C01819=1084.866,371.145,-96.496,176.864,26.563,154.394
C01820=1084.871,371.355,-96.527,176.867,26.567,154.395
C01821=1084.877,371.565,-96.559,176.870,26.572,154.396
C01822=1084.882,371.775,-96.590,176.873,26.578,154.397
C01823=1084.888,372.022,-96.627,176.876,26.584,154.398
C01824=1084.894,372.269,-96.664,176.880,26.590,154.399
C01825=1084.900,372.516,-96.701,176.883,26.596,154.400
C01826=1084.906,372.763,-96.738,176.886,26.603,154.401
C01827=1084.913,373.011,-96.775,176.890,26.609,154.403
C01828=1084.919,373.257,-96.812,176.892,26.615,154.404
C01829=1084.925,373.504,-96.849,176.896,26.621,154.405
C01830=1084.932,373.752,-96.885,176.900,26.627,154.406
C01831=1084.937,373.998,-96.923,176.902,26.633,154.407
C01832=1084.943,374.246,-96.960,176.906,26.640,154.408
C01833=1084.949,374.493,-96.997,176.909,26.646,154.409
C01834=1084.956,374.740,-97.035,176.913,26.652,154.410
C01835=1084.962,374.988,-97.072,176.916,26.658,154.412
C01836=1084.968,375.234,-97.109,176.919,26.665,154.413
C01837=1084.974,375.481,-97.146,176.923,26.672,154.414
C01838=1084.980,375.728,-97.184,176.925,26.678,154.415
C01839=1084.986,375.975,-97.220,176.929,26.684,154.416
C01840=1084.993,376.223,-97.258,176.933,26.690,154.417
C01841=1084.998,376.469,-97.296,176.936,26.697,154.418
C01842=1085.004,376.717,-97.333,176.939,26.703,154.420
C01843=1085.011,376.963,-97.370,176.942,26.709,154.421
C01844=1085.016,377.210,-97.407,176.946,26.716,154.422
C01845=1085.023,377.458,-97.445,176.948,26.722,154.423
C01846=1085.029,377.705,-97.483,176.952,26.729,154.424
C01847=1085.035,377.952,-97.520,176.955,26.736,154.426
C01848=1085.041,378.198,-97.557,176.959,26.742,154.427
C01849=1085.047,378.446,-97.595,176.962,26.748,154.428
C01850=1085.053,378.693,-97.633,176.965,26.755,154.429
C01851=1085.060,378.940,-97.670,176.969,26.761,154.430
C01852=1085.066,379.187,-97.708,176.972,26.768,154.431
C01853=1085.072,379.434,-97.745,176.976,26.775,154.433
C01854=1085.078,379.681,-97.783,176.979,26.781,154.434
C01855=1085.084,379.928,-97.821,176.982,26.788,154.435
C01856=1085.091,380.174,-97.859,176.986,26.795,154.436
C01857=1085.097,380.422,-97.896,176.989,26.801,154.438
C01858=1085.103,380.669,-97.934,176.993,26.808,154.439
C01859=1085.109,380.916,-97.971,176.995,26.814,154.440
C01860=1085.115,381.163,-98.009,176.999,26.821,154.441
C01861=1085.122,381.410,-98.047,177.002,26.828,154.443
C01862=1085.128,381.657,-98.084,177.006,26.834,154.444
C01863=1085.135,381.904,-98.123,177.009,26.841,154.445
C01864=1085.141,382.151,-98.160,177.012,26.847,154.446
C01865=1085.147,382.398,-98.198,177.016,26.854,154.447
C01866=1085.153,382.645,-98.236,177.019,26.861,154.449
C01867=1085.159,382.891,-98.275,177.022,26.868,154.450
C01868=1085.165,383.138,-98.312,177.026,26.875,154.451
C01869=1085.172,383.385,-98.351,177.030,26.882,154.453
C01870=1085.178,383.632,-98.388,177.032,26.888,154.454
C01871=1085.182,383.856,-98.423,177.036,26.895,154.455
C01872=1085.188,384.080,-98.458,177.038,26.901,154.456
C01873=1085.194,384.304,-98.492,177.042,26.908,154.457
C01874=1085.199,384.527,-98.527,177.045,26.914,154.459
C01875=1085.205,384.752,-98.562,177.047,26.920,154.460
C01876=1085.211,384.975,-98.596,177.051,26.926,154.461
C01877=1085.217,385.199,-98.631,177.054,26.932,154.462
C01878=1085.222,385.423,-98.666,177.057,26.939,154.463
C01879=1085.228,385.671,-98.704,177.061,26.946,154.465
C01880=1085.234,385.917,-98.742,177.063,26.953,154.466
C01881=1085.241,386.164,-98.780,177.067,26.960,154.467
C01882=1085.247,386.410,-98.819,177.070,26.967,154.469
C01883=1085.254,386.658,-98.857,177.074,26.974,154.470
C01884=1085.260,386.904,-98.895,177.077,26.981,154.471
C01885=1085.266,387.152,-98.934,177.081,26.988,154.473
C01886=1085.271,387.399,-98.972,177.084,26.995,154.474
C01887=1085.278,387.645,-99.011,177.088,27.003,154.475
C01888=1085.284,387.891,-99.049,177.091,27.010,154.477
C01889=1085.291,388.139,-99.087,177.095,27.017,154.478
C01890=1085.296,388.385,-99.126,177.098,27.024,154.479
C01891=1085.303,388.633,-99.165,177.101,27.031,154.481
C01892=1085.310,388.880,-99.203,177.105,27.038,154.482
C01893=1085.316,389.126,-99.242,177.108,27.045,154.484
C01894=1085.322,389.373,-99.280,177.111,27.053,154.485
C01895=1085.328,389.620,-99.319,177.114,27.060,154.486
C01896=1085.335,389.866,-99.358,177.118,27.067,154.488
C01897=1085.341,390.114,-99.396,177.121,27.075,154.489
C01898=1085.347,390.360,-99.434,177.125,27.082,154.491
C01899=1085.354,390.607,-99.474,177.128,27.089,154.492
C01900=1085.360,390.854,-99.513,177.132,27.096,154.493
C01901=1085.367,391.100,-99.551,177.135,27.104,154.495
C01902=1085.372,391.348,-99.590,177.139,27.111,154.496
C01903=1085.379,391.595,-99.629,177.142,27.119,154.498
C01904=1085.386,391.841,-99.668,177.146,27.126,154.499
C01905=1085.391,392.088,-99.707,177.149,27.133,154.500
C01906=1085.398,392.335,-99.746,177.152,27.141,154.502
C01907=1085.404,392.582,-99.785,177.156,27.148,154.503
C01908=1085.411,392.828,-99.823,177.159,27.156,154.505
C01909=1085.417,393.075,-99.863,177.163,27.163,154.506
C01910=1085.423,393.322,-99.902,177.166,27.171,154.508
C01911=1085.429,393.569,-99.941,177.170,27.179,154.509
C01912=1085.436,393.815,-99.980,177.173,27.186,154.511
C01913=1085.442,394.062,-100.019,177.176,27.194,154.512
C01914=1085.449,394.309,-100.058,177.180,27.201,154.514
C01915=1085.455,394.556,-100.097,177.183,27.209,154.515
C01916=1085.461,394.803,-100.136,177.187,27.217,154.517
C01917=1085.467,395.049,-100.176,177.191,27.225,154.518
C01918=1085.474,395.296,-100.215,177.194,27.232,154.520
C01919=1085.480,395.543,-100.254,177.198,27.240,154.521
C01920=1085.486,395.790,-100.294,177.201,27.248,154.523
C01921=1085.493,396.037,-100.332,177.205,27.256,154.524
C01922=1085.499,396.283,-100.373,177.208,27.264,154.526
C01923=1085.505,396.530,-100.412,177.211,27.271,154.527
C01924=1085.511,396.777,-100.451,177.215,27.279,154.529
C01925=1085.518,397.023,-100.491,177.218,27.287,154.530
C01926=1085.524,397.270,-100.530,177.222,27.295,154.532
C01927=1085.530,397.501,-100.566,177.225,27.302,154.533
C01928=1085.536,397.732,-100.604,177.229,27.310,154.535
C01929=1085.542,397.963,-100.640,177.231,27.317,154.536
C01930=1085.548,398.194,-100.678,177.235,27.325,154.538
C01931=1085.554,398.424,-100.715,177.238,27.332,154.539
C01932=1085.560,398.655,-100.752,177.242,27.339,154.541
C01933=1085.566,398.886,-100.789,177.245,27.347,154.542
C01934=1085.572,399.116,-100.826,177.248,27.354,154.544
C01935=1085.578,399.363,-100.866,177.252,27.363,154.545
C01936=1085.585,399.610,-100.905,177.255,27.371,154.547
C01937=1085.591,399.856,-100.945,177.258,27.379,154.549
C01938=1085.597,400.103,-100.985,177.262,27.387,154.550
C01939=1085.604,400.350,-101.025,177.265,27.395,154.552
C01940=1085.610,400.596,-101.065,177.269,27.404,154.553
C01941=1085.616,400.844,-101.104,177.272,27.411,154.555
C01942=1085.622,401.090,-101.145,177.276,27.420,154.557
C01943=1085.629,401.337,-101.185,177.280,27.428,154.558
C01944=1085.635,401.584,-101.224,177.283,27.437,154.560
C01945=1085.641,401.830,-101.264,177.286,27.445,154.562
C01946=1085.648,402.077,-101.305,177.290,27.453,154.563
C01947=1085.655,402.324,-101.345,177.294,27.462,154.565
C01948=1085.661,402.571,-101.385,177.297,27.470,154.567
C01949=1085.667,402.817,-101.425,177.301,27.478,154.568
C01950=1085.673,403.064,-101.465,177.304,27.487,154.570
C01951=1085.680,403.311,-101.505,177.308,27.495,154.572
C01952=1085.686,403.557,-101.545,177.312,27.504,154.573
C01953=1085.693,403.804,-101.585,177.315,27.512,154.575
C01954=1085.700,404.051,-101.626,177.318,27.521,154.577
C01955=1085.706,404.297,-101.666,177.323,27.529,154.579
C01956=1085.712,404.544,-101.706,177.326,27.537,154.580
C01957=1085.719,404.790,-101.746,177.329,27.546,154.582
C01958=1085.725,405.037,-101.786,177.333,27.555,154.584
C01959=1085.731,405.283,-101.826,177.337,27.564,154.586
C01960=1085.738,405.531,-101.867,177.340,27.572,154.587
C01961=1085.745,405.777,-101.908,177.343,27.581,154.589
C01962=1085.751,406.023,-101.949,177.348,27.590,154.591
C01963=1085.757,406.270,-101.989,177.351,27.598,154.593
C01964=1085.764,406.517,-102.029,177.354,27.607,154.594
C01965=1085.771,406.764,-102.069,177.359,27.616,154.596
C01966=1085.776,407.010,-102.111,177.362,27.625,154.598
C01967=1085.783,407.256,-102.151,177.365,27.634,154.600
C01968=1085.790,407.504,-102.191,177.369,27.643,154.602
C01969=1085.797,407.750,-102.232,177.373,27.652,154.604
C01970=1085.802,407.996,-102.273,177.376,27.660,154.605
C01971=1085.809,408.244,-102.314,177.380,27.669,154.607
C01972=1085.815,408.490,-102.355,177.383,27.679,154.609
C01973=1085.821,408.736,-102.395,177.388,27.688,154.611
C01974=1085.828,408.982,-102.436,177.391,27.697,154.613
C01975=1085.834,409.230,-102.477,177.394,27.705,154.615
C01976=1085.841,409.476,-102.518,177.399,27.715,154.616
C01977=1085.847,409.722,-102.559,177.402,27.724,154.618
C01978=1085.854,409.969,-102.600,177.406,27.733,154.620
C01979=1085.860,410.216,-102.640,177.409,27.742,154.622
C01980=1085.867,410.462,-102.682,177.413,27.751,154.624
C01981=1085.874,410.708,-102.723,177.417,27.761,154.626
C01982=1085.879,410.955,-102.764,177.420,27.770,154.628
C01983=1085.886,411.187,-102.802,177.424,27.779,154.630
C01984=1085.892,411.418,-102.841,177.428,27.788,154.631
C01985=1085.898,411.649,-102.879,177.431,27.796,154.633
C01986=1085.904,411.882,-102.918,177.434,27.805,154.635
C01987=1085.910,412.113,-102.956,177.438,27.814,154.637
C01988=1085.917,412.344,-102.996,177.441,27.822,154.639
C01989=1085.923,412.576,-103.035,177.444,27.832,154.641
C01990=1085.929,412.807,-103.072,177.449,27.841,154.642
C01991=1085.935,413.054,-103.114,177.452,27.850,154.644
C01992=1085.942,413.300,-103.155,177.456,27.859,154.646
C01993=1085.948,413.547,-103.197,177.459,27.869,154.648
C01994=1085.956,413.793,-103.238,177.464,27.878,154.650
C01995=1085.962,414.040,-103.280,177.467,27.888,154.652
C01996=1085.969,414.286,-103.321,177.471,27.897,154.654
C01997=1085.975,414.532,-103.362,177.475,27.907,154.656
C01998=1085.982,414.779,-103.404,177.479,27.917,154.658
C01999=1085.988,415.025,-103.445,177.483,27.926,154.660
C02000=1085.995,415.272,-103.487,177.486,27.936,154.662
C02001=1086.002,415.519,-103.528,177.490,27.946,154.664
C02002=1086.008,415.765,-103.570,177.494,27.956,154.666
C02003=1086.015,416.011,-103.611,177.498,27.966,154.668
C02004=1086.022,416.258,-103.653,177.502,27.976,154.671
C02005=1086.028,416.504,-103.695,177.505,27.985,154.673
C02006=1086.035,416.751,-103.737,177.509,27.996,154.675
C02007=1086.041,416.997,-103.779,177.513,28.005,154.677
C02008=1086.048,417.243,-103.820,177.517,28.016,154.679
C02009=1086.055,417.490,-103.862,177.521,28.025,154.681
C02010=1086.061,417.736,-103.904,177.525,28.036,154.683
C02011=1086.067,417.983,-103.946,177.529,28.046,154.685
C02012=1086.074,418.229,-103.988,177.532,28.056,154.687
C02013=1086.080,418.475,-104.030,177.536,28.066,154.690
C02014=1086.087,418.721,-104.072,177.541,28.076,154.692
C02015=1086.094,418.968,-104.114,177.544,28.086,154.694
C02016=1086.101,419.214,-104.156,177.548,28.097,154.696
C02017=1086.107,419.460,-104.198,177.552,28.107,154.698
C02018=1086.114,419.707,-104.240,177.556,28.117,154.700
C02019=1086.121,419.954,-104.282,177.560,28.127,154.703
C02020=1086.127,420.200,-104.324,177.564,28.138,154.705
C02021=1086.134,420.445,-104.367,177.568,28.149,154.707
C02022=1086.140,420.692,-104.408,177.572,28.159,154.709
C02023=1086.147,420.939,-104.451,177.575,28.169,154.711
C02024=1086.154,421.185,-104.494,177.579,28.180,154.714
C02025=1086.162,421.431,-104.535,177.583,28.190,154.716
C02026=1086.168,421.677,-104.578,177.588,28.201,154.718
C02027=1086.174,421.923,-104.619,177.592,28.211,154.720
C02028=1086.181,422.170,-104.662,177.596,28.222,154.723
C02029=1086.188,422.416,-104.705,177.599,28.233,154.725
C02030=1086.194,422.663,-104.748,177.603,28.244,154.727
C02031=1086.201,422.909,-104.790,177.607,28.254,154.730
C02032=1086.208,423.155,-104.833,177.611,28.265,154.732
C02033=1086.215,423.401,-104.875,177.616,28.276,154.734
C02034=1086.221,423.647,-104.917,177.620,28.287,154.737
C02035=1086.228,423.893,-104.960,177.624,28.298,154.739
C02036=1086.234,424.140,-105.003,177.627,28.309,154.741
C02037=1086.241,424.386,-105.046,177.631,28.319,154.744
C02038=1086.248,424.632,-105.089,177.635,28.331,154.746
C02039=1086.259,425.045,-105.160,177.642,28.349,154.750
C02040=1086.271,425.458,-105.232,177.649,28.368,154.754
C02041=1086.282,425.871,-105.304,177.656,28.386,154.758
C02042=1086.293,426.284,-105.376,177.663,28.405,154.762
C02043=1086.300,426.529,-105.419,177.667,28.417,154.765
C02044=1086.307,426.775,-105.462,177.671,28.428,154.767
C02045=1086.313,427.022,-105.505,177.675,28.439,154.769
C02046=1086.320,427.268,-105.548,177.679,28.450,154.772
C02047=1086.327,427.514,-105.591,177.683,28.462,154.774
C02048=1086.334,427.760,-105.634,177.687,28.473,154.777
C02049=1086.341,428.006,-105.678,177.691,28.485,154.779
C02050=1086.348,428.253,-105.721,177.695,28.496,154.782
C02051=1086.356,428.498,-105.764,177.700,28.507,154.784
C02052=1086.362,428.745,-105.807,177.704,28.519,154.787
C02053=1086.369,428.991,-105.851,177.709,28.531,154.789
C02054=1086.375,429.237,-105.894,177.713,28.543,154.792
C02055=1086.382,429.482,-105.938,177.717,28.555,154.795
C02056=1086.389,429.729,-105.981,177.721,28.566,154.797
C02057=1086.396,429.974,-106.024,177.725,28.578,154.800
C02058=1086.403,430.221,-106.068,177.729,28.590,154.802
C02059=1086.410,430.467,-106.112,177.733,28.602,154.805
C02060=1086.416,430.713,-106.155,177.737,28.614,154.808
C02061=1086.423,430.958,-106.199,177.741,28.626,154.810
C02062=1086.430,431.204,-106.243,177.746,28.638,154.813
C02063=1086.437,431.451,-106.287,177.751,28.650,154.815
C02064=1086.444,431.697,-106.330,177.755,28.662,154.818
C02065=1086.450,431.943,-106.374,177.759,28.674,154.821
C02066=1086.458,432.188,-106.417,177.763,28.686,154.823
C02067=1086.465,432.435,-106.461,177.767,28.698,154.826
C02068=1086.472,432.681,-106.505,177.772,28.710,154.829
C02069=1086.478,432.927,-106.548,177.776,28.723,154.832
C02070=1086.485,433.173,-106.593,177.780,28.735,154.834
C02071=1086.492,433.419,-106.637,177.784,28.748,154.837
C02072=1086.499,433.664,-106.680,177.789,28.760,154.840
C02073=1086.506,433.911,-106.725,177.793,28.773,154.843
C02074=1086.513,434.156,-106.769,177.797,28.785,154.845
C02075=1086.521,434.468,-106.825,177.803,28.801,154.849
C02076=1086.530,434.780,-106.881,177.808,28.817,154.852
C02077=1086.539,435.092,-106.937,177.814,28.833,154.856
C02078=1086.548,435.404,-106.993,177.820,28.849,154.860
C02079=1086.555,435.649,-107.037,177.824,28.862,154.862
C02080=1086.561,435.895,-107.081,177.829,28.875,154.865
C02081=1086.569,436.141,-107.126,177.833,28.888,154.868
C02082=1086.575,436.387,-107.171,177.837,28.901,154.871
C02083=1086.583,436.633,-107.214,177.842,28.914,154.874
C02084=1086.590,436.878,-107.259,177.846,28.926,154.877
C02085=1086.597,437.124,-107.304,177.850,28.939,154.880
C02086=1086.604,437.370,-107.349,177.855,28.953,154.883
C02087=1086.611,437.616,-107.393,177.859,28.966,154.886
C02088=1086.618,437.862,-107.437,177.864,28.979,154.888
C02089=1086.625,438.108,-107.482,177.868,28.992,154.891
C02090=1086.632,438.353,-107.527,177.872,29.005,154.894
C02091=1086.639,438.584,-107.568,177.876,29.018,154.897
C02092=1086.646,438.814,-107.610,177.881,29.030,154.900
C02093=1086.652,439.044,-107.653,177.886,29.043,154.903
C02094=1086.658,439.274,-107.694,177.890,29.056,154.906
C02095=1086.666,439.505,-107.737,177.894,29.068,154.909
C02096=1086.672,439.735,-107.778,177.898,29.081,154.911
C02097=1086.679,439.966,-107.821,177.902,29.093,154.914
C02098=1086.686,440.196,-107.863,177.907,29.106,154.917
C02099=1086.693,440.442,-107.908,177.911,29.120,154.920
C02100=1086.700,440.687,-107.953,177.916,29.134,154.923
C02101=1086.707,440.933,-107.998,177.920,29.147,154.926
C02102=1086.715,441.179,-108.043,177.925,29.161,154.930
C02103=1086.721,441.424,-108.088,177.930,29.175,154.933
C02104=1086.728,441.670,-108.133,177.934,29.189,154.936
C02105=1086.736,441.916,-108.179,177.939,29.203,154.939
C02106=1086.743,442.162,-108.224,177.943,29.217,154.942
C02107=1086.750,442.407,-108.268,177.948,29.231,154.945
C02108=1086.756,442.653,-108.315,177.952,29.245,154.949
C02109=1086.764,442.898,-108.360,177.957,29.260,154.952
C02110=1086.771,443.144,-108.405,177.962,29.274,154.955
C02111=1086.778,443.389,-108.451,177.966,29.288,154.958
C02112=1086.785,443.635,-108.496,177.971,29.302,154.962
C02113=1086.793,443.881,-108.542,177.976,29.317,154.965
C02114=1086.800,444.127,-108.588,177.980,29.331,154.968
C02115=1086.807,444.373,-108.633,177.985,29.346,154.972
C02116=1086.815,444.618,-108.679,177.991,29.360,154.975
C02117=1086.821,444.863,-108.724,177.995,29.374,154.978
C02118=1086.829,445.109,-108.770,178.000,29.389,154.981
C02119=1086.836,445.354,-108.816,178.004,29.404,154.985
C02120=1086.843,445.600,-108.862,178.008,29.418,154.988
C02121=1086.851,445.845,-108.908,178.012,29.433,154.992
C02122=1086.858,446.091,-108.954,178.016,29.448,154.995
C02123=1086.865,446.336,-108.999,178.019,29.462,154.999
C02124=1086.872,446.582,-109.046,178.022,29.477,155.002
C02125=1086.880,446.828,-109.091,178.025,29.491,155.005
C02126=1086.887,447.073,-109.138,178.029,29.506,155.009
C02127=1086.894,447.319,-109.183,178.032,29.520,155.012
C02128=1086.901,447.565,-109.229,178.034,29.535,155.016
C02129=1086.908,447.810,-109.276,178.036,29.549,155.019
C02130=1086.916,448.056,-109.321,178.038,29.563,155.023
C02131=1086.923,448.301,-109.368,178.040,29.578,155.027
C02132=1086.931,448.546,-109.414,178.043,29.593,155.030
C02133=1086.938,448.793,-109.461,178.044,29.607,155.034
C02134=1086.946,449.038,-109.506,178.045,29.621,155.037
C02135=1086.952,449.283,-109.553,178.046,29.636,155.041
C02136=1086.960,449.527,-109.599,178.048,29.650,155.044
C02137=1086.969,449.773,-109.645,178.049,29.664,155.048
C02138=1086.980,450.019,-109.689,178.050,29.676,155.051
C02139=1086.604,450.011,-109.889,178.013,29.864,155.102
C02140=1086.592,449.765,-109.845,178.012,29.851,155.098
C02141=1086.583,449.520,-109.798,178.010,29.837,155.095
C02142=1086.576,449.275,-109.753,178.009,29.823,155.091
C02143=1086.568,449.031,-109.707,178.007,29.808,155.088
C02144=1086.561,448.785,-109.661,178.006,29.794,155.084
C02145=1086.554,448.540,-109.614,178.005,29.780,155.081
C02146=1086.546,448.294,-109.568,178.002,29.765,155.077
C02147=1086.539,448.048,-109.521,178.000,29.750,155.074
C02148=1086.531,447.803,-109.475,177.998,29.736,155.070
C02149=1086.524,447.557,-109.429,177.995,29.721,155.066
C02150=1086.516,447.312,-109.383,177.993,29.707,155.063
C02151=1086.510,447.066,-109.337,177.990,29.693,155.060
C02152=1086.503,446.820,-109.291,177.987,29.678,155.056
C02153=1086.495,446.576,-109.244,177.983,29.663,155.053
C02154=1086.488,446.330,-109.198,177.980,29.649,155.049
C02155=1086.480,446.084,-109.152,177.977,29.634,155.046
C02156=1086.473,445.839,-109.106,177.973,29.619,155.042
C02157=1086.466,445.593,-109.060,177.969,29.605,155.039
C02158=1086.459,445.347,-109.014,177.964,29.590,155.035
C02159=1086.451,445.102,-108.969,177.960,29.576,155.032
C02160=1086.443,444.857,-108.923,177.955,29.561,155.029
C02161=1086.437,444.611,-108.877,177.950,29.546,155.025
C02162=1086.429,444.365,-108.832,177.946,29.532,155.022
C02163=1086.422,444.119,-108.786,177.941,29.517,155.019
C02164=1086.415,443.874,-108.740,177.935,29.503,155.015
C02165=1086.407,443.628,-108.694,177.931,29.489,155.012
C02166=1086.401,443.383,-108.648,177.926,29.474,155.009
C02167=1086.393,443.137,-108.603,177.921,29.460,155.005
C02168=1086.386,442.892,-108.558,177.917,29.446,155.002
C02169=1086.378,442.646,-108.513,177.912,29.431,154.999
C02170=1086.372,442.400,-108.467,177.907,29.417,154.996
C02171=1086.365,442.155,-108.421,177.902,29.403,154.993
C02172=1086.357,441.909,-108.376,177.897,29.389,154.989
C02173=1086.350,441.664,-108.331,177.893,29.375,154.986
C02174=1086.343,441.417,-108.285,177.888,29.361,154.983
C02175=1086.336,441.172,-108.241,177.884,29.347,154.980
C02176=1086.329,440.927,-108.195,177.879,29.333,154.977
C02177=1086.321,440.680,-108.150,177.874,29.320,154.974
C02178=1086.314,440.434,-108.105,177.869,29.306,154.971
C02179=1086.307,440.190,-108.060,177.865,29.292,154.967
C02180=1086.301,439.966,-108.018,177.861,29.280,154.965
C02181=1086.294,439.742,-107.978,177.857,29.267,154.962
C02182=1086.288,439.519,-107.937,177.852,29.255,154.959
C02183=1086.281,439.295,-107.896,177.848,29.243,154.956
C02184=1086.275,439.072,-107.855,177.844,29.231,154.954
C02185=1086.267,438.849,-107.815,177.839,29.218,154.951
C02186=1086.261,438.626,-107.774,177.836,29.206,154.948
C02187=1086.255,438.402,-107.733,177.832,29.194,154.945
C02188=1086.247,438.156,-107.688,177.826,29.181,154.942
C02189=1086.241,437.911,-107.644,177.822,29.168,154.939
C02190=1086.233,437.665,-107.599,177.818,29.155,154.936
C02191=1086.227,437.420,-107.554,177.813,29.141,154.933
C02192=1086.220,437.173,-107.510,177.809,29.128,154.931
C02193=1086.212,436.927,-107.465,177.804,29.115,154.928
C02194=1086.206,436.681,-107.421,177.800,29.102,154.925
C02195=1086.199,436.436,-107.376,177.795,29.089,154.922
C02196=1086.191,436.190,-107.333,177.790,29.076,154.919
C02197=1086.184,435.944,-107.288,177.786,29.063,154.916
C02198=1086.177,435.698,-107.243,177.782,29.050,154.913
C02199=1086.171,435.452,-107.199,177.777,29.037,154.910
C02200=1086.163,435.206,-107.154,177.773,29.025,154.907
C02201=1086.157,434.961,-107.110,177.768,29.012,154.905
C02202=1086.150,434.714,-107.065,177.764,28.999,154.902
C02203=1086.142,434.469,-107.021,177.759,28.987,154.899
C02204=1086.136,434.223,-106.978,177.755,28.974,154.896
C02205=1086.129,433.977,-106.933,177.751,28.961,154.893
C02206=1086.122,433.731,-106.889,177.747,28.949,154.891
C02207=1086.115,433.485,-106.845,177.742,28.936,154.888
C02208=1086.107,433.240,-106.801,177.738,28.924,154.885
C02209=1086.101,432.994,-106.757,177.733,28.912,154.882
C02210=1086.095,432.748,-106.713,177.729,28.899,154.880
C02211=1086.088,432.501,-106.669,177.725,28.887,154.877
C02212=1086.080,432.255,-106.626,177.720,28.875,154.874
C02213=1086.074,432.010,-106.581,177.716,28.863,154.872
C02214=1086.066,431.764,-106.537,177.712,28.851,154.869
C02215=1086.059,431.518,-106.493,177.707,28.838,154.866
C02216=1086.052,431.272,-106.450,177.703,28.826,154.863
C02217=1086.045,431.025,-106.406,177.699,28.815,154.861
C02218=1086.039,430.779,-106.362,177.694,28.802,154.858
C02219=1086.032,430.534,-106.319,177.690,28.790,154.856
C02220=1086.025,430.288,-106.275,177.686,28.778,154.853
C02221=1086.018,430.042,-106.232,177.681,28.766,154.850
C02222=1086.011,429.795,-106.188,177.677,28.755,154.848
C02223=1086.004,429.550,-106.144,177.673,28.743,154.845
C02224=1085.998,429.303,-106.101,177.669,28.731,154.843
C02225=1085.991,429.057,-106.058,177.665,28.720,154.840
C02226=1085.984,428.811,-106.014,177.661,28.708,154.838
C02227=1085.977,428.566,-105.971,177.656,28.696,154.835
C02228=1085.970,428.318,-105.927,177.652,28.685,154.832
C02229=1085.963,428.073,-105.884,177.648,28.673,154.830
C02230=1085.956,427.827,-105.841,177.643,28.661,154.827
C02231=1085.949,427.581,-105.798,177.639,28.650,154.825
C02232=1085.943,427.335,-105.754,177.634,28.639,154.822
C02233=1085.936,427.089,-105.712,177.630,28.627,154.820
C02234=1085.929,426.843,-105.669,177.626,28.616,154.817
C02235=1085.922,426.596,-105.625,177.622,28.604,154.815
C02236=1085.915,426.356,-105.583,177.619,28.593,154.813
C02237=1085.908,426.116,-105.542,177.614,28.582,154.810
C02238=1085.902,425.877,-105.499,177.610,28.571,154.808
C02239=1085.896,425.636,-105.458,177.606,28.561,154.806
C02240=1085.889,425.397,-105.415,177.602,28.549,154.803
C02241=1085.882,425.157,-105.374,177.598,28.539,154.801
C02242=1085.876,424.917,-105.333,177.594,28.528,154.799
C02243=1085.869,424.677,-105.290,177.590,28.517,154.796
C02244=1085.862,424.431,-105.248,177.586,28.506,154.794
C02245=1085.855,424.184,-105.205,177.582,28.495,154.791
C02246=1085.849,423.938,-105.163,177.577,28.484,154.789
C02247=1085.842,423.692,-105.119,177.574,28.473,154.787
C02248=1085.835,423.446,-105.076,177.570,28.462,154.784
C02249=1085.828,423.200,-105.034,177.566,28.452,154.782
C02250=1085.822,422.953,-104.991,177.562,28.441,154.780
C02251=1085.815,422.707,-104.949,177.557,28.430,154.777
C02252=1085.808,422.461,-104.906,177.553,28.419,154.775
C02253=1085.802,422.215,-104.863,177.549,28.408,154.773
C02254=1085.796,421.969,-104.821,177.546,28.398,154.771
C02255=1085.789,421.722,-104.778,177.542,28.387,154.768
C02256=1085.781,421.476,-104.737,177.537,28.376,154.766
C02257=1085.775,421.229,-104.694,177.533,28.366,154.764
C02258=1085.768,420.983,-104.652,177.529,28.355,154.761
C02259=1085.761,420.737,-104.609,177.526,28.345,154.759
C02260=1085.754,420.491,-104.567,177.522,28.334,154.757
C02261=1085.748,420.244,-104.525,177.517,28.324,154.755
C02262=1085.741,419.998,-104.483,177.513,28.314,154.753
C02263=1085.734,419.752,-104.440,177.510,28.303,154.750
C02264=1085.724,419.343,-104.370,177.503,28.286,154.747
C02265=1085.712,418.933,-104.301,177.497,28.269,154.743
C02266=1085.702,418.525,-104.231,177.490,28.252,154.740
C02267=1085.690,418.115,-104.161,177.484,28.235,154.736
C02268=1085.684,417.869,-104.119,177.479,28.225,154.734
C02269=1085.677,417.623,-104.077,177.475,28.215,154.732
C02270=1085.670,417.376,-104.035,177.472,28.205,154.730
C02271=1085.664,417.130,-103.993,177.467,28.195,154.727
C02272=1085.657,416.884,-103.951,177.463,28.184,154.725
C02273=1085.650,416.637,-103.910,177.460,28.175,154.723
C02274=1085.644,416.391,-103.868,177.456,28.164,154.721
C02275=1085.637,416.144,-103.826,177.452,28.154,154.719
C02276=1085.631,415.898,-103.784,177.448,28.145,154.717
C02277=1085.624,415.652,-103.743,177.444,28.135,154.715
C02278=1085.618,415.405,-103.701,177.441,28.125,154.713
C02279=1085.610,415.159,-103.659,177.436,28.115,154.711
C02280=1085.604,414.913,-103.618,177.432,28.106,154.709
C02281=1085.597,414.666,-103.576,177.429,28.096,154.707
C02282=1085.591,414.420,-103.535,177.425,28.086,154.705
C02283=1085.584,414.173,-103.493,177.421,28.077,154.703
C02284=1085.577,413.926,-103.452,177.417,28.067,154.701
C02285=1085.571,413.680,-103.410,177.414,28.058,154.699
C02286=1085.564,413.434,-103.369,177.409,28.048,154.697
C02287=1085.558,413.187,-103.328,177.406,28.039,154.695
C02288=1085.551,412.941,-103.286,177.402,28.029,154.693
C02289=1085.545,412.695,-103.245,177.399,28.020,154.691
C02290=1085.537,412.448,-103.204,177.394,28.010,154.689
C02291=1085.531,412.202,-103.162,177.391,28.000,154.687
C02292=1085.523,411.900,-103.112,177.386,27.989,154.684
C02293=1085.515,411.598,-103.062,177.381,27.978,154.682
C02294=1085.506,411.297,-103.011,177.376,27.966,154.680
C02295=1085.500,410.996,-102.961,177.372,27.955,154.677
C02296=1085.492,410.749,-102.920,177.368,27.945,154.676
C02297=1085.487,410.502,-102.879,177.365,27.936,154.674
C02298=1085.479,410.256,-102.838,177.360,27.927,154.672
C02299=1085.473,410.010,-102.797,177.357,27.918,154.670
C02300=1085.467,409.763,-102.756,177.354,27.908,154.668
C02301=1085.460,409.517,-102.715,177.349,27.899,154.666
C02302=1085.454,409.270,-102.674,177.346,27.890,154.664
C02303=1085.447,409.023,-102.633,177.342,27.881,154.662
C02304=1085.440,408.777,-102.592,177.339,27.872,154.660
C02305=1085.435,408.530,-102.552,177.335,27.863,154.658
C02306=1085.428,408.283,-102.511,177.331,27.854,154.657
C02307=1085.422,408.037,-102.470,177.328,27.845,154.655
C02308=1085.415,407.790,-102.429,177.324,27.836,154.653
C02309=1085.409,407.545,-102.389,177.320,27.827,154.651
C02310=1085.402,407.297,-102.347,177.317,27.818,154.649
C02311=1085.396,407.051,-102.307,177.312,27.809,154.647
C02312=1085.389,406.805,-102.266,177.309,27.800,154.646
C02313=1085.382,406.557,-102.226,177.306,27.791,154.644
C02314=1085.377,406.311,-102.185,177.302,27.782,154.642
C02315=1085.370,406.065,-102.144,177.298,27.774,154.640
C02316=1085.364,405.818,-102.104,177.295,27.765,154.638
C02317=1085.357,405.571,-102.064,177.291,27.756,154.637
C02318=1085.350,405.324,-102.024,177.287,27.747,154.635
C02319=1085.345,405.078,-101.983,177.284,27.739,154.633
C02320=1085.338,404.831,-101.943,177.280,27.730,154.631
C02321=1085.331,404.584,-101.902,177.277,27.722,154.630
C02322=1085.325,404.337,-101.862,177.272,27.713,154.628
C02323=1085.318,404.091,-101.821,177.269,27.704,154.626
C02324=1085.312,403.845,-101.781,177.266,27.696,154.624
C02325=1085.305,403.598,-101.741,177.262,27.687,154.623
C02326=1085.299,403.352,-101.701,177.258,27.679,154.621
C02327=1085.292,403.104,-101.661,177.255,27.670,154.619
C02328=1085.286,402.858,-101.621,177.251,27.662,154.618
C02329=1085.280,402.611,-101.581,177.248,27.654,154.616
C02330=1085.273,402.365,-101.540,177.243,27.645,154.614
C02331=1085.267,402.118,-101.500,177.240,27.636,154.612
C02332=1085.260,401.872,-101.460,177.237,27.628,154.611
C02333=1085.254,401.625,-101.420,177.233,27.620,154.609
C02334=1085.247,401.377,-101.380,177.230,27.612,154.607
C02335=1085.241,401.131,-101.340,177.226,27.604,154.606
C02336=1085.235,400.884,-101.300,177.222,27.595,154.604
C02337=1085.228,400.638,-101.260,177.219,27.587,154.603
C02338=1085.222,400.390,-101.220,177.215,27.579,154.601
C02339=1085.216,400.144,-101.180,177.212,27.570,154.599
C02340=1085.209,399.897,-101.140,177.208,27.562,154.598
C02341=1085.203,399.651,-101.101,177.205,27.554,154.596
C02342=1085.196,399.404,-101.061,177.201,27.545,154.594
C02343=1085.190,399.158,-101.021,177.197,27.538,154.593
C02344=1085.184,398.926,-100.984,177.195,27.530,154.591
C02345=1085.178,398.694,-100.947,177.191,27.523,154.590
C02346=1085.172,398.464,-100.910,177.188,27.515,154.588
C02347=1085.166,398.233,-100.872,177.184,27.508,154.587
C02348=1085.160,398.001,-100.835,177.181,27.500,154.585
C02349=1085.154,397.769,-100.799,177.178,27.493,154.584
C02350=1085.148,397.538,-100.761,177.175,27.485,154.582
C02351=1085.143,397.307,-100.724,177.171,27.478,154.581
C02352=1085.136,397.061,-100.685,177.168,27.470,154.579
C02353=1085.129,396.814,-100.645,177.164,27.462,154.578
C02354=1085.123,396.567,-100.606,177.161,27.454,154.576
C02355=1085.117,396.320,-100.566,177.157,27.446,154.575
C02356=1085.110,396.074,-100.527,177.154,27.438,154.573
C02357=1085.104,395.826,-100.487,177.150,27.431,154.572
C02358=1085.098,395.579,-100.448,177.147,27.423,154.570
C02359=1085.091,395.333,-100.409,177.144,27.415,154.568
C02360=1085.085,395.087,-100.369,177.140,27.407,154.567
C02361=1085.079,394.840,-100.330,177.137,27.400,154.565
C02362=1085.073,394.593,-100.291,177.133,27.392,154.564
C02363=1085.067,394.346,-100.251,177.130,27.384,154.562
C02364=1085.060,394.099,-100.212,177.126,27.377,154.561
C02365=1085.054,393.852,-100.173,177.122,27.368,154.559
C02366=1085.047,393.606,-100.135,177.118,27.361,154.558
C02367=1085.041,393.358,-100.095,177.115,27.354,154.557
C02368=1085.035,393.112,-100.056,177.111,27.346,154.555
C02369=1085.028,392.865,-100.016,177.108,27.338,154.554
C02370=1085.022,392.619,-99.978,177.105,27.330,154.552
C02371=1085.016,392.372,-99.938,177.101,27.323,154.551
C02372=1085.009,392.124,-99.900,177.097,27.316,154.549
C02373=1085.004,391.878,-99.861,177.095,27.308,154.548
C02374=1084.997,391.631,-99.822,177.092,27.301,154.546
C02375=1084.990,391.384,-99.783,177.088,27.293,154.545
C02376=1084.984,391.137,-99.744,177.085,27.286,154.543
C02377=1084.978,390.891,-99.706,177.081,27.279,154.542
C02378=1084.971,390.644,-99.667,177.078,27.271,154.540
C02379=1084.965,390.397,-99.627,177.074,27.264,154.539
C02380=1084.959,390.150,-99.589,177.070,27.257,154.538
C02381=1084.952,389.903,-99.551,177.067,27.249,154.536
C02382=1084.946,389.657,-99.512,177.064,27.242,154.535
C02383=1084.940,389.410,-99.473,177.060,27.235,154.534
C02384=1084.934,389.163,-99.435,177.057,27.227,154.532
C02385=1084.927,388.916,-99.396,177.053,27.220,154.531
C02386=1084.921,388.670,-99.357,177.049,27.213,154.529
C02387=1084.914,388.422,-99.319,177.046,27.206,154.528
C02388=1084.908,388.175,-99.280,177.042,27.199,154.527
C02389=1084.902,387.929,-99.241,177.039,27.191,154.525
C02390=1084.895,387.682,-99.203,177.035,27.184,154.524
C02391=1084.889,387.436,-99.165,177.032,27.177,154.523
C02392=1084.883,387.188,-99.127,177.028,27.170,154.521
C02393=1084.877,386.942,-99.088,177.026,27.163,154.520
C02394=1084.871,386.694,-99.049,177.022,27.156,154.518
C02395=1084.864,386.448,-99.011,177.019,27.149,154.517
C02396=1084.858,386.201,-98.973,177.015,27.142,154.516
C02397=1084.851,385.954,-98.934,177.012,27.135,154.514
C02398=1084.845,385.707,-98.896,177.008,27.128,154.513
C02399=1084.840,385.461,-98.857,177.005,27.120,154.512
C02400=1084.834,385.236,-98.823,177.002,27.114,154.511
C02401=1084.828,385.012,-98.788,176.998,27.108,154.509
C02402=1084.823,384.787,-98.753,176.996,27.101,154.508
C02403=1084.816,384.563,-98.718,176.993,27.095,154.507
C02404=1084.811,384.337,-98.684,176.989,27.089,154.506
C02405=1084.806,384.114,-98.649,176.987,27.082,154.505
C02406=1084.800,383.890,-98.614,176.983,27.076,154.503
C02407=1084.794,383.665,-98.580,176.980,27.070,154.502
C02408=1084.789,383.418,-98.541,176.977,27.063,154.501
C02409=1084.782,383.171,-98.503,176.973,27.056,154.500
C02410=1084.776,382.924,-98.466,176.971,27.049,154.498
C02411=1084.770,382.677,-98.428,176.967,27.042,154.497
C02412=1084.764,382.431,-98.389,176.963,27.036,154.496
C02413=1084.758,382.184,-98.351,176.960,27.029,154.495
C02414=1084.751,381.936,-98.313,176.956,27.022,154.493
C02415=1084.745,381.690,-98.275,176.953,27.015,154.492
C02416=1084.738,381.442,-98.238,176.950,27.009,154.491
C02417=1084.732,381.196,-98.200,176.947,27.002,154.489
C02418=1084.726,380.949,-98.162,176.943,26.995,154.488
C02419=1084.720,380.702,-98.124,176.939,26.988,154.487
C02420=1084.714,380.455,-98.086,176.937,26.982,154.486
C02421=1084.707,380.207,-98.048,176.933,26.975,154.485
C02422=1084.701,379.961,-98.011,176.930,26.969,154.483
C02423=1084.695,379.714,-97.974,176.926,26.962,154.482
C02424=1084.689,379.466,-97.936,176.923,26.955,154.481
C02425=1084.683,379.219,-97.898,176.920,26.949,154.480
C02426=1084.677,378.973,-97.860,176.916,26.942,154.479
C02427=1084.670,378.726,-97.823,176.913,26.936,154.477
C02428=1084.664,378.479,-97.785,176.909,26.929,154.476
C02429=1084.658,378.231,-97.748,176.906,26.923,154.475
C02430=1084.652,377.985,-97.710,176.903,26.916,154.474
C02431=1084.646,377.737,-97.672,176.899,26.909,154.472
C02432=1084.639,377.491,-97.635,176.896,26.903,154.471
C02433=1084.633,377.243,-97.598,176.893,26.897,154.470
C02434=1084.627,376.997,-97.560,176.889,26.890,154.469
C02435=1084.621,376.749,-97.522,176.886,26.884,154.468
C02436=1084.615,376.502,-97.486,176.883,26.878,154.467
C02437=1084.609,376.255,-97.448,176.880,26.871,154.465
C02438=1084.603,376.008,-97.411,176.876,26.865,154.464
C02439=1084.596,375.762,-97.374,176.872,26.858,154.463
C02440=1084.590,375.514,-97.336,176.870,26.852,154.462
C02441=1084.584,375.267,-97.299,176.866,26.845,154.461
C02442=1084.578,375.020,-97.261,176.863,26.839,154.460
C02443=1084.572,374.773,-97.224,176.860,26.833,154.458
C02444=1084.566,374.526,-97.187,176.856,26.826,154.457
C02445=1084.561,374.279,-97.150,176.853,26.820,154.456
C02446=1084.554,374.031,-97.113,176.850,26.814,154.455
C02447=1084.548,373.784,-97.075,176.846,26.807,154.454
C02448=1084.541,373.537,-97.039,176.843,26.801,154.453
C02449=1084.536,373.290,-97.002,176.840,26.795,154.452
C02450=1084.529,373.044,-96.964,176.836,26.789,154.450
C02451=1084.524,372.796,-96.927,176.833,26.783,154.449
C02452=1084.517,372.548,-96.891,176.830,26.776,154.448
C02453=1084.511,372.302,-96.853,176.826,26.770,154.447
C02454=1084.504,372.055,-96.816,176.823,26.764,154.446
C02455=1084.498,371.808,-96.780,176.820,26.758,154.445
C02456=1084.494,371.597,-96.748,176.817,26.753,154.444
C02457=1084.488,371.386,-96.717,176.814,26.748,154.443
C02458=1084.483,371.176,-96.686,176.812,26.742,154.442
C02459=1084.477,370.967,-96.654,176.809,26.737,154.441
C02460=1084.471,370.756,-96.622,176.806,26.732,154.440
C02461=1084.467,370.546,-96.591,176.803,26.727,154.439
C02462=1084.462,370.336,-96.560,176.800,26.722,154.438
C02463=1084.456,370.125,-96.528,176.797,26.716,154.438
C02464=1084.450,369.878,-96.492,176.794,26.710,154.437
C02465=1084.444,369.630,-96.455,176.791,26.705,154.435
C02466=1084.438,369.383,-96.418,176.787,26.699,154.434
C02467=1084.432,369.136,-96.382,176.785,26.692,154.433
C02468=1084.426,368.889,-96.345,176.781,26.686,154.432
C02469=1084.420,368.642,-96.308,176.777,26.680,154.431
C02470=1084.414,368.395,-96.271,176.775,26.674,154.430
C02471=1084.408,368.148,-96.235,176.771,26.668,154.429
C02472=1084.401,367.900,-96.198,176.768,26.663,154.428
C02473=1084.396,367.653,-96.161,176.764,26.657,154.427
C02474=1084.389,367.406,-96.125,176.761,26.651,154.426
C02475=1084.383,367.158,-96.089,176.758,26.645,154.425
C02476=1084.378,366.911,-96.052,176.754,26.639,154.424
C02477=1084.371,366.664,-96.016,176.752,26.633,154.423
C02478=1084.365,366.417,-95.979,176.748,26.627,154.422
C02479=1084.359,366.171,-95.943,176.745,26.621,154.421
C02480=1084.354,365.923,-95.907,176.742,26.615,154.420
C02481=1084.348,365.676,-95.871,176.738,26.609,154.419
C02482=1084.341,365.428,-95.834,176.735,26.603,154.418
C02483=1084.335,365.181,-95.798,176.732,26.598,154.417
C02484=1084.330,364.933,-95.761,176.729,26.592,154.416
C02485=1084.323,364.686,-95.725,176.725,26.586,154.415
C02486=1084.317,364.439,-95.688,176.722,26.581,154.414
C02487=1084.311,364.192,-95.653,176.719,26.575,154.413
C02488=1084.305,363.945,-95.616,176.716,26.569,154.412
C02489=1084.299,363.697,-95.580,176.712,26.563,154.411
C02490=1084.292,363.450,-95.544,176.709,26.557,154.410
C02491=1084.287,363.204,-95.508,176.706,26.552,154.409
C02492=1084.281,362.956,-95.472,176.702,26.546,154.408
C02493=1084.274,362.709,-95.436,176.699,26.541,154.407
C02494=1084.268,362.461,-95.400,176.696,26.535,154.406
C02495=1084.262,362.214,-95.364,176.693,26.529,154.405
C02496=1084.257,361.966,-95.327,176.689,26.523,154.404
C02497=1084.250,361.719,-95.291,176.686,26.518,154.403
C02498=1084.244,361.471,-95.255,176.683,26.512,154.402
C02499=1084.239,361.224,-95.220,176.680,26.507,154.401
C02500=1084.232,360.977,-95.183,176.676,26.501,154.400
C02501=1084.226,360.730,-95.148,176.673,26.496,154.399
C02502=1084.220,360.482,-95.112,176.670,26.490,154.398
C02503=1084.214,360.235,-95.075,176.667,26.484,154.397
C02504=1084.209,359.988,-95.040,176.663,26.479,154.396
C02505=1084.202,359.741,-95.005,176.661,26.473,154.395
C02506=1084.196,359.494,-94.968,176.657,26.467,154.394
C02507=1084.190,359.246,-94.933,176.654,26.462,154.393
C02508=1084.183,358.998,-94.897,176.650,26.457,154.392
C02509=1084.178,358.751,-94.862,176.648,26.451,154.391
C02510=1084.172,358.504,-94.826,176.644,26.446,154.391
C02511=1084.166,358.256,-94.789,176.641,26.440,154.390
C02512=1084.156,357.852,-94.732,176.636,26.432,154.388
C02513=1084.146,357.447,-94.673,176.630,26.422,154.387
C02514=1084.136,357.042,-94.615,176.625,26.413,154.385
C02515=1084.126,356.638,-94.557,176.620,26.405,154.384
C02516=1084.120,356.390,-94.521,176.616,26.399,154.383
C02517=1084.114,356.143,-94.485,176.614,26.394,154.382
C02518=1084.108,355.896,-94.451,176.611,26.389,154.381
C02519=1084.102,355.648,-94.415,176.607,26.383,154.380
C02520=1084.096,355.400,-94.380,176.604,26.378,154.379
C02521=1084.091,355.153,-94.345,176.601,26.372,154.378
C02522=1084.085,354.905,-94.309,176.598,26.367,154.377
C02523=1084.078,354.658,-94.274,176.594,26.361,154.376
C02524=1084.072,354.411,-94.238,176.591,26.357,154.376
C02525=1084.066,354.163,-94.203,176.588,26.351,154.375
C02526=1084.060,353.916,-94.168,176.585,26.346,154.374
C02527=1084.054,353.669,-94.132,176.582,26.340,154.373
C02528=1084.048,353.421,-94.097,176.578,26.335,154.372
C02529=1084.042,353.173,-94.061,176.575,26.330,154.371
C02530=1084.036,352.926,-94.027,176.572,26.325,154.370
C02531=1084.030,352.679,-93.991,176.569,26.320,154.369
C02532=1084.024,352.431,-93.957,176.566,26.314,154.368
C02533=1084.018,352.184,-93.921,176.562,26.309,154.368
C02534=1084.012,351.936,-93.885,176.559,26.304,154.367
C02535=1084.006,351.689,-93.851,176.556,26.299,154.366
C02536=1084.000,351.441,-93.816,176.553,26.293,154.365
C02537=1083.994,351.194,-93.781,176.550,26.289,154.364
C02538=1083.988,350.946,-93.746,176.546,26.283,154.363
C02539=1083.982,350.699,-93.711,176.543,26.278,154.363
C02540=1083.976,350.452,-93.675,176.540,26.273,154.362
C02541=1083.970,350.204,-93.641,176.537,26.268,154.361
C02542=1083.964,349.957,-93.606,176.534,26.262,154.360
C02543=1083.958,349.709,-93.571,176.531,26.258,154.359
C02544=1083.953,349.462,-93.536,176.527,26.252,154.358
C02545=1083.946,349.214,-93.501,176.524,26.247,154.357
C02546=1083.941,348.967,-93.466,176.522,26.242,154.357
C02547=1083.934,348.719,-93.432,176.518,26.237,154.356
C02548=1083.929,348.472,-93.396,176.515,26.232,154.355
C02549=1083.922,348.224,-93.362,176.512,26.227,154.354
C02550=1083.916,347.977,-93.327,176.508,26.222,154.353
C02551=1083.910,347.729,-93.292,176.505,26.217,154.353
C02552=1083.905,347.482,-93.258,176.503,26.212,154.352
C02553=1083.898,347.234,-93.222,176.499,26.207,154.351
C02554=1083.893,346.987,-93.188,176.496,26.202,154.350
C02555=1083.886,346.739,-93.154,176.493,26.197,154.349
C02556=1083.881,346.492,-93.118,176.489,26.192,154.349
C02557=1083.874,346.244,-93.084,176.487,26.187,154.348
C02558=1083.869,345.996,-93.049,176.484,26.182,154.347
C02559=1083.863,345.749,-93.015,176.480,26.177,154.346
C02560=1083.857,345.502,-92.980,176.477,26.172,154.345
C02561=1083.851,345.254,-92.945,176.474,26.167,154.344
C02562=1083.845,345.006,-92.911,176.470,26.162,154.344
C02563=1083.839,344.759,-92.877,176.467,26.157,154.343
C02564=1083.830,344.357,-92.821,176.462,26.149,154.342
C02565=1083.819,343.955,-92.765,176.457,26.141,154.340
C02566=1083.810,343.553,-92.709,176.452,26.133,154.339
C02567=1083.801,343.151,-92.654,176.447,26.125,154.338
C02568=1083.794,342.903,-92.619,176.444,26.120,154.337
C02569=1083.788,342.656,-92.585,176.441,26.115,154.336
C02570=1083.782,342.409,-92.551,176.437,26.110,154.335
C02571=1083.777,342.160,-92.516,176.434,26.106,154.335
C02572=1083.771,341.913,-92.482,176.432,26.101,154.334
C02573=1083.765,341.666,-92.448,176.429,26.096,154.333
C02574=1083.759,341.418,-92.414,176.425,26.091,154.332
C02575=1083.753,341.171,-92.380,176.422,26.086,154.332
C02576=1083.747,340.923,-92.345,176.419,26.082,154.331
C02577=1083.740,340.675,-92.311,176.416,26.077,154.330
C02578=1083.735,340.428,-92.277,176.413,26.072,154.329
C02579=1083.729,340.181,-92.243,176.410,26.067,154.329
C02580=1083.723,339.932,-92.209,176.407,26.063,154.328
C02581=1083.717,339.685,-92.175,176.404,26.058,154.327
C02582=1083.712,339.437,-92.141,176.400,26.053,154.326
C02583=1083.706,339.190,-92.106,176.397,26.048,154.326
C02584=1083.699,338.942,-92.072,176.394,26.043,154.325
C02585=1083.694,338.694,-92.039,176.391,26.039,154.324
C02586=1083.688,338.447,-92.005,176.388,26.034,154.324
C02587=1083.682,338.200,-91.971,176.385,26.029,154.323
C02588=1083.676,337.951,-91.937,176.382,26.024,154.322
C02589=1083.670,337.704,-91.903,176.379,26.020,154.321
C02590=1083.664,337.456,-91.869,176.376,26.015,154.320
C02591=1083.658,337.209,-91.835,176.372,26.010,154.320
C02592=1083.652,336.961,-91.801,176.369,26.005,154.319
C02593=1083.646,336.713,-91.767,176.366,26.001,154.318
C02594=1083.640,336.466,-91.734,176.363,25.997,154.318
C02595=1083.634,336.218,-91.700,176.361,25.992,154.317
C02596=1083.628,335.970,-91.667,176.357,25.987,154.316
C02597=1083.622,335.722,-91.632,176.354,25.982,154.315
C02598=1083.616,335.475,-91.599,176.351,25.978,154.315
C02599=1083.611,335.227,-91.565,176.348,25.973,154.314
C02600=1083.605,334.979,-91.532,176.345,25.969,154.313
C02601=1083.598,334.732,-91.498,176.341,25.964,154.313
C02602=1083.593,334.485,-91.465,176.338,25.959,154.312
C02603=1083.586,334.237,-91.430,176.335,25.955,154.311
C02604=1083.581,333.989,-91.397,176.332,25.950,154.311
C02605=1083.575,333.741,-91.363,176.330,25.946,154.310
C02606=1083.569,333.493,-91.330,176.327,25.941,154.309
C02607=1083.563,333.246,-91.297,176.323,25.936,154.309
C02608=1083.557,332.999,-91.263,176.320,25.932,154.308
C02609=1083.552,332.751,-91.230,176.317,25.927,154.307
C02610=1083.546,332.503,-91.196,176.314,25.923,154.306
C02611=1083.540,332.255,-91.162,176.311,25.918,154.306
C02612=1083.534,332.008,-91.129,176.308,25.914,154.305
C02613=1083.528,331.759,-91.096,176.304,25.909,154.304
C02614=1083.522,331.511,-91.062,176.301,25.905,154.304
C02615=1083.516,331.264,-91.029,176.298,25.900,154.303
C02616=1083.506,330.857,-90.975,176.293,25.893,154.302
C02617=1083.496,330.449,-90.919,176.289,25.886,154.301
C02618=1083.486,330.042,-90.865,176.284,25.878,154.300
C02619=1083.477,329.634,-90.811,176.278,25.871,154.299
C02620=1083.470,329.387,-90.777,176.276,25.867,154.298
C02621=1083.464,329.139,-90.744,176.273,25.862,154.297
C02622=1083.458,328.891,-90.711,176.270,25.858,154.297
C02623=1083.452,328.644,-90.678,176.267,25.854,154.296
C02624=1083.447,328.396,-90.645,176.263,25.849,154.295
C02625=1083.440,328.148,-90.612,176.260,25.845,154.295
C02626=1083.435,327.900,-90.579,176.257,25.840,154.294
C02627=1083.428,327.653,-90.546,176.254,25.836,154.293
C02628=1083.423,327.405,-90.513,176.251,25.832,154.293
C02629=1083.417,327.157,-90.480,176.248,25.827,154.292
C02630=1083.411,326.909,-90.447,176.245,25.823,154.291
C02631=1083.405,326.662,-90.414,176.242,25.818,154.291
C02632=1083.398,326.414,-90.381,176.239,25.815,154.290
C02633=1083.393,326.166,-90.349,176.236,25.810,154.290
C02634=1083.387,325.918,-90.316,176.232,25.805,154.289
C02635=1083.381,325.670,-90.283,176.229,25.801,154.288
C02636=1083.375,325.422,-90.250,176.226,25.797,154.288
C02637=1083.369,325.175,-90.217,176.223,25.792,154.287
C02638=1083.363,324.927,-90.184,176.220,25.788,154.286
C02639=1083.357,324.679,-90.152,176.217,25.784,154.286
C02640=1083.352,324.431,-90.118,176.215,25.780,154.285
C02641=1083.345,324.183,-90.086,176.212,25.775,154.284
C02642=1083.339,323.936,-90.053,176.209,25.771,154.284
C02643=1083.334,323.687,-90.020,176.206,25.767,154.283
C02644=1083.328,323.440,-89.988,176.203,25.763,154.283
C02645=1083.322,323.193,-89.955,176.200,25.758,154.282
C02646=1083.316,322.945,-89.922,176.197,25.754,154.281
C02647=1083.310,322.697,-89.890,176.194,25.749,154.281
C02648=1083.304,322.449,-89.857,176.191,25.746,154.280
C02649=1083.298,322.201,-89.824,176.188,25.741,154.279
C02650=1083.293,321.954,-89.792,176.184,25.736,154.279
C02651=1083.287,321.706,-89.759,176.181,25.732,154.278
C02652=1083.281,321.457,-89.727,176.178,25.728,154.278
C02653=1083.275,321.210,-89.694,176.175,25.724,154.277
C02654=1083.269,320.962,-89.661,176.172,25.719,154.276
C02655=1083.264,320.714,-89.629,176.169,25.715,154.276
C02656=1083.258,320.467,-89.596,176.166,25.711,154.275
C02657=1083.252,320.219,-89.564,176.163,25.707,154.274
C02658=1083.246,319.971,-89.531,176.160,25.703,154.274
C02659=1083.240,319.722,-89.499,176.157,25.698,154.273
C02660=1083.235,319.476,-89.466,176.155,25.694,154.273
C02661=1083.229,319.227,-89.434,176.151,25.690,154.272
C02662=1083.223,318.979,-89.402,176.149,25.686,154.271
C02663=1083.218,318.732,-89.369,176.146,25.681,154.271
C02664=1083.212,318.484,-89.337,176.143,25.677,154.270
C02665=1083.206,318.236,-89.305,176.140,25.673,154.269
C02666=1083.200,317.988,-89.272,176.137,25.668,154.269
C02667=1083.195,317.740,-89.240,176.134,25.665,154.268
C02668=1083.186,317.326,-89.186,176.129,25.657,154.267
C02669=1083.175,316.912,-89.132,176.124,25.650,154.266
C02670=1083.166,316.498,-89.079,176.119,25.643,154.265
C02671=1083.156,316.084,-89.024,176.115,25.636,154.264
C02672=1083.151,315.836,-88.992,176.112,25.632,154.264
C02673=1083.145,315.588,-88.961,176.109,25.628,154.263
C02674=1083.139,315.340,-88.929,176.106,25.624,154.262
C02675=1083.134,315.092,-88.895,176.103,25.620,154.262
C02676=1083.128,314.845,-88.864,176.100,25.616,154.261
C02677=1083.122,314.596,-88.832,176.097,25.611,154.261
C02678=1083.115,314.348,-88.800,176.094,25.607,154.260
C02679=1083.110,314.101,-88.769,176.091,25.604,154.259
C02680=1083.104,313.853,-88.737,176.088,25.600,154.259
C02681=1083.098,313.604,-88.705,176.085,25.595,154.258
C02682=1083.092,313.356,-88.673,176.082,25.591,154.258
C02683=1083.086,313.110,-88.641,176.079,25.587,154.257
C02684=1083.080,312.861,-88.609,176.076,25.583,154.257
C02685=1083.074,312.613,-88.577,176.073,25.580,154.256
C02686=1083.068,312.366,-88.545,176.070,25.575,154.256
C02687=1083.062,312.118,-88.514,176.067,25.571,154.255
C02688=1083.056,311.870,-88.482,176.064,25.567,154.254
C02689=1083.050,311.622,-88.450,176.061,25.563,154.254
C02690=1083.044,311.374,-88.418,176.058,25.559,154.253
C02691=1083.038,311.127,-88.387,176.055,25.556,154.253
C02692=1083.032,310.878,-88.356,176.052,25.551,154.252
C02693=1083.027,310.630,-88.324,176.049,25.547,154.252
C02694=1083.021,310.382,-88.292,176.046,25.543,154.251
C02695=1083.014,310.134,-88.260,176.043,25.539,154.251
C02696=1083.009,309.887,-88.229,176.040,25.535,154.250
C02697=1083.003,309.639,-88.197,176.038,25.532,154.250
C02698=1082.997,309.391,-88.166,176.034,25.528,154.249
C02699=1082.991,309.143,-88.134,176.032,25.523,154.248
C02700=1082.986,308.895,-88.103,176.029,25.520,154.248
C02701=1082.980,308.647,-88.071,176.026,25.516,154.247
C02702=1082.974,308.400,-88.040,176.023,25.512,154.247
C02703=1082.968,308.151,-88.008,176.019,25.508,154.246
C02704=1082.963,307.903,-87.977,176.016,25.504,154.246
C02705=1082.956,307.655,-87.945,176.013,25.500,154.245
C02706=1082.951,307.408,-87.913,176.010,25.496,154.245
C02707=1082.944,307.160,-87.882,176.007,25.492,154.244
C02708=1082.939,306.912,-87.851,176.005,25.488,154.243
C02709=1082.933,306.664,-87.819,176.001,25.484,154.243
C02710=1082.927,306.416,-87.788,175.999,25.480,154.242
C02711=1082.922,306.168,-87.757,175.996,25.476,154.242
C02712=1082.916,305.920,-87.725,175.993,25.472,154.241
C02713=1082.910,305.672,-87.695,175.990,25.468,154.241
C02714=1082.904,305.424,-87.663,175.987,25.464,154.240
C02715=1082.898,305.177,-87.632,175.984,25.460,154.240
C02716=1082.893,304.929,-87.601,175.981,25.456,154.239
C02717=1082.887,304.680,-87.569,175.978,25.453,154.239
C02718=1082.881,304.433,-87.538,175.975,25.449,154.238
C02719=1082.875,304.185,-87.507,175.972,25.445,154.238
C02720=1082.865,303.774,-87.455,175.968,25.438,154.237
C02721=1082.856,303.363,-87.403,175.963,25.431,154.236
C02722=1082.846,302.951,-87.351,175.958,25.425,154.235
C02723=1082.837,302.540,-87.300,175.954,25.419,154.234
C02724=1082.831,302.292,-87.269,175.951,25.415,154.233
C02725=1082.826,302.044,-87.238,175.948,25.411,154.233
C02726=1082.820,301.796,-87.206,175.945,25.407,154.232
C02727=1082.814,301.548,-87.176,175.942,25.403,154.232
C02728=1082.809,301.300,-87.145,175.939,25.399,154.231
C02729=1082.803,301.053,-87.114,175.936,25.395,154.231
C02730=1082.797,300.804,-87.082,175.934,25.391,154.230
C02731=1082.791,300.556,-87.052,175.931,25.387,154.230
C02732=1082.786,300.308,-87.021,175.928,25.383,154.229
C02733=1082.780,300.061,-86.990,175.925,25.380,154.229
C02734=1082.774,299.812,-86.959,175.922,25.376,154.228
C02735=1082.768,299.564,-86.928,175.919,25.372,154.228
C02736=1082.763,299.316,-86.897,175.916,25.368,154.227
C02737=1082.757,299.069,-86.866,175.914,25.364,154.227
C02738=1082.752,298.821,-86.835,175.911,25.360,154.226
C02739=1082.746,298.572,-86.805,175.908,25.356,154.226
C02740=1082.741,298.324,-86.774,175.905,25.352,154.225
C02741=1082.735,298.076,-86.743,175.902,25.348,154.224
C02742=1082.729,297.829,-86.712,175.899,25.344,154.224
C02743=1082.724,297.581,-86.681,175.896,25.341,154.223
C02744=1082.717,297.332,-86.651,175.893,25.337,154.223
C02745=1082.711,297.085,-86.620,175.890,25.333,154.222
C02746=1082.706,296.837,-86.590,175.887,25.329,154.222
C02747=1082.701,296.589,-86.559,175.884,25.325,154.221
C02748=1082.694,296.340,-86.528,175.881,25.322,154.221
C02749=1082.688,296.092,-86.498,175.879,25.318,154.220
C02750=1082.682,295.844,-86.468,175.876,25.314,154.220
C02751=1082.677,295.597,-86.437,175.873,25.310,154.219
C02752=1082.672,295.348,-86.406,175.870,25.307,154.219
C02753=1082.665,295.100,-86.376,175.867,25.303,154.218
C02754=1082.659,294.852,-86.345,175.864,25.299,154.218
C02755=1082.654,294.604,-86.315,175.862,25.295,154.217
C02756=1082.648,294.356,-86.285,175.859,25.292,154.217
C02757=1082.642,294.109,-86.254,175.856,25.288,154.216
C02758=1082.636,293.860,-86.225,175.853,25.284,154.216
C02759=1082.631,293.611,-86.193,175.850,25.281,154.216
C02760=1082.625,293.364,-86.163,175.848,25.277,154.215
C02761=1082.619,293.116,-86.133,175.845,25.273,154.214
C02762=1082.613,292.868,-86.102,175.842,25.269,154.214
C02763=1082.607,292.620,-86.072,175.838,25.266,154.214
C02764=1082.602,292.372,-86.042,175.835,25.262,154.213
C02765=1082.596,292.124,-86.012,175.833,25.258,154.212
C02766=1082.590,291.876,-85.982,175.830,25.255,154.212
C02767=1082.584,291.627,-85.951,175.827,25.251,154.212
C02768=1082.578,291.380,-85.920,175.824,25.247,154.211
C02769=1082.573,291.131,-85.891,175.822,25.244,154.211
C02770=1082.567,290.883,-85.860,175.819,25.240,154.210
C02771=1082.561,290.636,-85.830,175.816,25.236,154.210
C02772=1082.552,290.238,-85.781,175.812,25.230,154.209
C02773=1082.543,289.842,-85.734,175.807,25.224,154.208
C02774=1082.534,289.444,-85.686,175.803,25.218,154.207
C02775=1082.524,289.047,-85.638,175.798,25.212,154.207
C02776=1082.519,288.799,-85.607,175.795,25.208,154.206
C02777=1082.513,288.551,-85.577,175.792,25.205,154.206
C02778=1082.507,288.303,-85.547,175.790,25.201,154.205
C02779=1082.501,288.055,-85.518,175.787,25.198,154.205
C02780=1082.495,287.807,-85.488,175.784,25.194,154.204
C02781=1082.489,287.559,-85.458,175.781,25.190,154.204
C02782=1082.484,287.311,-85.428,175.779,25.187,154.203
C02783=1082.478,287.063,-85.398,175.775,25.183,154.203
C02784=1082.473,286.815,-85.368,175.772,25.179,154.202
C02785=1082.466,286.567,-85.338,175.769,25.176,154.202
C02786=1082.461,286.319,-85.309,175.767,25.172,154.201
C02787=1082.455,286.070,-85.279,175.764,25.169,154.201
C02788=1082.449,285.822,-85.249,175.761,25.165,154.200
C02789=1082.444,285.574,-85.219,175.758,25.161,154.200
C02790=1082.437,285.326,-85.189,175.756,25.158,154.200
C02791=1082.432,285.078,-85.160,175.753,25.154,154.199
C02792=1082.426,284.829,-85.130,175.750,25.150,154.199
C02793=1082.420,284.582,-85.100,175.747,25.146,154.198
C02794=1082.415,284.333,-85.070,175.745,25.143,154.198
C02795=1082.409,284.085,-85.041,175.742,25.139,154.197
C02796=1082.403,283.837,-85.011,175.739,25.136,154.197
C02797=1082.397,283.589,-84.981,175.737,25.132,154.196
C02798=1082.392,283.340,-84.951,175.733,25.129,154.196
C02799=1082.385,283.092,-84.922,175.731,25.125,154.195
C02800=1082.380,282.844,-84.893,175.727,25.121,154.195
C02801=1082.374,282.596,-84.862,175.725,25.118,154.194
C02802=1082.369,282.348,-84.833,175.722,25.114,154.194
C02803=1082.363,282.100,-84.804,175.719,25.110,154.193
C02804=1082.357,281.852,-84.774,175.717,25.107,154.193
C02805=1082.352,281.603,-84.745,175.714,25.103,154.192
C02806=1082.345,281.356,-84.715,175.711,25.099,154.192
C02807=1082.340,281.107,-84.685,175.708,25.095,154.192
C02808=1082.334,280.859,-84.656,175.706,25.092,154.191
C02809=1082.328,280.611,-84.627,175.703,25.089,154.191
C02810=1082.323,280.362,-84.597,175.700,25.085,154.190
C02811=1082.318,280.114,-84.568,175.698,25.082,154.190
C02812=1082.311,279.866,-84.539,175.695,25.078,154.189
C02813=1082.306,279.618,-84.509,175.691,25.074,154.189
C02814=1082.300,279.370,-84.480,175.689,25.071,154.188
C02815=1082.294,279.121,-84.451,175.686,25.067,154.188
C02816=1082.288,278.873,-84.421,175.683,25.064,154.188
C02817=1082.282,278.625,-84.392,175.681,25.061,154.187
C02818=1082.277,278.377,-84.363,175.678,25.057,154.187
C02819=1082.271,278.129,-84.334,175.675,25.053,154.186
C02820=1082.265,277.881,-84.304,175.672,25.049,154.186
C02821=1082.259,277.632,-84.275,175.670,25.046,154.185
C02822=1082.253,277.384,-84.246,175.667,25.042,154.185
C02823=1082.248,277.136,-84.216,175.664,25.038,154.184
C02824=1082.239,276.749,-84.171,175.660,25.033,154.184
C02825=1082.230,276.361,-84.126,175.656,25.028,154.183
C02826=1082.221,275.973,-84.080,175.651,25.022,154.182
C02827=1082.212,275.587,-84.035,175.647,25.017,154.182
C02828=1082.207,275.338,-84.006,175.644,25.013,154.181
C02829=1082.200,275.090,-83.977,175.641,25.009,154.181
C02830=1082.195,274.842,-83.948,175.639,25.006,154.180
C02831=1082.189,274.594,-83.919,175.636,25.003,154.180
C02832=1082.184,274.345,-83.890,175.633,24.999,154.179
C02833=1082.178,274.097,-83.861,175.631,24.996,154.179
C02834=1082.172,273.850,-83.832,175.628,24.992,154.179
C02835=1082.167,273.601,-83.803,175.625,24.988,154.178
C02836=1082.161,273.352,-83.774,175.623,24.985,154.178
C02837=1082.154,273.104,-83.745,175.620,24.981,154.177
C02838=1082.150,272.856,-83.717,175.616,24.978,154.177
C02839=1082.143,272.608,-83.688,175.614,24.974,154.176
C02840=1082.137,272.360,-83.659,175.611,24.971,154.176
C02841=1082.131,272.111,-83.630,175.608,24.967,154.176
C02842=1082.126,271.863,-83.601,175.606,24.964,154.175
C02843=1082.120,271.614,-83.573,175.603,24.960,154.175
C02844=1082.114,271.366,-83.544,175.601,24.957,154.174
C02845=1082.109,271.119,-83.515,175.598,24.953,154.174
C02846=1082.103,270.870,-83.486,175.595,24.949,154.173
C02847=1082.097,270.622,-83.457,175.593,24.946,154.173
C02848=1082.092,270.374,-83.429,175.590,24.943,154.172
C02849=1082.085,270.126,-83.400,175.587,24.939,154.172
C02850=1082.080,269.876,-83.371,175.585,24.936,154.171
C02851=1082.075,269.629,-83.342,175.581,24.932,154.171
C02852=1082.069,269.380,-83.314,175.579,24.929,154.171
C02853=1082.063,269.132,-83.286,175.576,24.926,154.170
C02854=1082.057,268.884,-83.257,175.573,24.922,154.170
C02855=1082.051,268.635,-83.229,175.571,24.918,154.169
C02856=1082.046,268.387,-83.199,175.568,24.915,154.169
C02857=1082.040,268.139,-83.171,175.565,24.911,154.169
C02858=1082.034,267.890,-83.143,175.563,24.908,154.168
C02859=1082.029,267.643,-83.114,175.560,24.904,154.168
C02860=1082.023,267.394,-83.086,175.558,24.901,154.167
C02861=1082.017,267.145,-83.058,175.554,24.898,154.167
C02862=1082.011,266.898,-83.029,175.551,24.894,154.166
C02863=1082.005,266.649,-83.001,175.549,24.891,154.166
C02864=1082.000,266.401,-82.973,175.546,24.887,154.166
C02865=1081.994,266.152,-82.944,175.544,24.884,154.165
C02866=1081.988,265.904,-82.915,175.541,24.880,154.165
C02867=1081.982,265.656,-82.887,175.538,24.877,154.164
C02868=1081.977,265.407,-82.858,175.536,24.873,154.164
C02869=1081.972,265.159,-82.830,175.533,24.870,154.163
C02870=1081.966,264.911,-82.801,175.531,24.866,154.163
C02871=1081.960,264.663,-82.773,175.528,24.863,154.163
C02872=1081.954,264.414,-82.745,175.525,24.860,154.162
C02873=1081.949,264.166,-82.717,175.522,24.856,154.162
C02874=1081.943,263.917,-82.689,175.519,24.852,154.161
C02875=1081.936,263.669,-82.661,175.517,24.849,154.161
C02876=1081.927,263.284,-82.617,175.513,24.844,154.160
C02877=1081.918,262.900,-82.574,175.509,24.839,154.160
C02878=1081.910,262.517,-82.530,175.504,24.834,154.159
C02879=1081.900,262.132,-82.487,175.501,24.828,154.158
C02880=1081.894,261.883,-82.459,175.498,24.825,154.158
C02881=1081.889,261.635,-82.431,175.495,24.821,154.158
C02882=1081.883,261.386,-82.403,175.492,24.818,154.157
C02883=1081.877,261.139,-82.375,175.489,24.815,154.157
C02884=1081.871,260.890,-82.347,175.487,24.811,154.156
C02885=1081.865,260.641,-82.319,175.484,24.808,154.156
C02886=1081.860,260.393,-82.291,175.482,24.805,154.156
C02887=1081.853,260.145,-82.263,175.479,24.801,154.155
C02888=1081.848,259.897,-82.235,175.477,24.798,154.155
C02889=1081.842,259.648,-82.207,175.474,24.795,154.154
C02890=1081.837,259.400,-82.179,175.471,24.791,154.154
C02891=1081.830,259.151,-82.151,175.468,24.788,154.154
C02892=1081.825,258.903,-82.124,175.465,24.784,154.153
C02893=1081.819,258.655,-82.096,175.463,24.781,154.153
C02894=1081.813,258.406,-82.068,175.460,24.777,154.152
C02895=1081.807,258.158,-82.040,175.458,24.774,154.152
C02896=1081.802,257.909,-82.012,175.455,24.771,154.151
C02897=1081.796,257.661,-81.985,175.453,24.767,154.151
C02898=1081.790,257.412,-81.957,175.450,24.764,154.151
C02899=1081.784,257.164,-81.929,175.448,24.761,154.150
C02900=1081.779,256.915,-81.901,175.445,24.757,154.150
C02901=1081.773,256.667,-81.874,175.441,24.754,154.149
C02902=1081.767,256.419,-81.846,175.439,24.751,154.149
C02903=1081.761,256.170,-81.818,175.436,24.747,154.149
C02904=1081.755,255.923,-81.790,175.434,24.744,154.148
C02905=1081.750,255.674,-81.763,175.431,24.740,154.148
C02906=1081.744,255.425,-81.735,175.429,24.737,154.147
C02907=1081.738,255.177,-81.707,175.426,24.733,154.147
C02908=1081.733,254.928,-81.680,175.424,24.730,154.147
C02909=1081.727,254.680,-81.652,175.421,24.726,154.146
C02910=1081.722,254.432,-81.625,175.419,24.723,154.146
C02911=1081.716,254.183,-81.597,175.415,24.720,154.145
C02912=1081.710,253.935,-81.569,175.413,24.717,154.145
C02913=1081.705,253.686,-81.542,175.410,24.713,154.145
C02914=1081.699,253.438,-81.514,175.408,24.710,154.144
C02915=1081.693,253.189,-81.487,175.405,24.706,154.144
C02916=1081.687,252.941,-81.459,175.403,24.703,154.143
C02917=1081.682,252.693,-81.433,175.400,24.699,154.143
C02918=1081.676,252.444,-81.404,175.398,24.696,154.142
C02919=1081.671,252.196,-81.377,175.395,24.692,154.142
C02920=1081.665,251.948,-81.350,175.393,24.689,154.142
C02921=1081.659,251.698,-81.322,175.390,24.686,154.141
C02922=1081.653,251.451,-81.295,175.387,24.683,154.141
C02923=1081.648,251.202,-81.267,175.384,24.679,154.140
C02924=1081.642,250.954,-81.240,175.382,24.676,154.140
C02925=1081.636,250.705,-81.212,175.379,24.672,154.139
C02926=1081.631,250.456,-81.185,175.377,24.669,154.139
C02927=1081.625,250.208,-81.158,175.374,24.665,154.139
C02928=1081.617,249.822,-81.116,175.370,24.660,154.138
C02929=1081.607,249.434,-81.073,175.366,24.654,154.137
C02930=1081.599,249.047,-81.031,175.362,24.649,154.137
C02931=1081.590,248.661,-80.988,175.359,24.644,154.136
C02932=1081.585,248.412,-80.961,175.356,24.640,154.136
C02933=1081.579,248.163,-80.934,175.353,24.637,154.135
C02934=1081.574,247.914,-80.906,175.350,24.634,154.135
C02935=1081.568,247.666,-80.879,175.348,24.631,154.134
C02936=1081.563,247.418,-80.852,175.345,24.627,154.134
C02937=1081.557,247.169,-80.825,175.343,24.623,154.134
C02938=1081.552,246.921,-80.798,175.340,24.620,154.133
C02939=1081.545,246.672,-80.771,175.338,24.617,154.133
C02940=1081.539,246.424,-80.744,175.335,24.613,154.132
C02941=1081.534,246.175,-80.716,175.333,24.610,154.132
C02942=1081.528,245.927,-80.690,175.330,24.606,154.132
C02943=1081.523,245.678,-80.663,175.328,24.603,154.131
C02944=1081.518,245.430,-80.636,175.325,24.600,154.131
C02945=1081.511,245.181,-80.609,175.322,24.597,154.130
C02946=1081.506,244.932,-80.582,175.320,24.593,154.130
C02947=1081.500,244.684,-80.555,175.317,24.590,154.130
C02948=1081.495,244.435,-80.528,175.315,24.587,154.129
C02949=1081.489,244.188,-80.501,175.312,24.583,154.129
C02950=1081.483,243.939,-80.474,175.310,24.580,154.128
C02951=1081.478,243.691,-80.447,175.307,24.576,154.128
C02952=1081.472,243.442,-80.420,175.305,24.573,154.128
C02953=1081.466,243.193,-80.393,175.302,24.570,154.127
C02954=1081.460,242.945,-80.367,175.300,24.566,154.127
C02955=1081.455,242.696,-80.339,175.297,24.563,154.126
C02956=1081.449,242.448,-80.313,175.294,24.560,154.126
C02957=1081.444,242.199,-80.287,175.292,24.557,154.126
C02958=1081.438,241.950,-80.260,175.289,24.553,154.125
C02959=1081.432,241.702,-80.234,175.287,24.550,154.125
C02960=1081.426,241.454,-80.207,175.284,24.546,154.124
C02961=1081.420,241.205,-80.180,175.282,24.543,154.124
C02962=1081.414,240.956,-80.153,175.279,24.540,154.124
C02963=1081.408,240.708,-80.127,175.277,24.536,154.123
C02964=1081.403,240.460,-80.100,175.275,24.533,154.123
C02965=1081.398,240.211,-80.073,175.271,24.530,154.122
C02966=1081.392,239.962,-80.047,175.269,24.527,154.122
C02967=1081.386,239.714,-80.020,175.266,24.523,154.122
C02968=1081.381,239.465,-79.993,175.264,24.520,154.121
C02969=1081.375,239.217,-79.967,175.262,24.517,154.121
C02970=1081.369,238.968,-79.940,175.259,24.513,154.120
C02971=1081.364,238.720,-79.914,175.257,24.510,154.120
C02972=1081.358,238.471,-79.888,175.254,24.506,154.120
C02973=1081.352,238.223,-79.861,175.252,24.503,154.119
C02974=1081.346,237.974,-79.834,175.249,24.500,154.119
C02975=1081.341,237.725,-79.808,175.247,24.496,154.118
C02976=1081.335,237.477,-79.782,175.244,24.493,154.118
C02977=1081.329,237.229,-79.755,175.241,24.490,154.118
C02978=1081.324,236.980,-79.729,175.239,24.486,154.117
C02979=1081.318,236.731,-79.702,175.236,24.483,154.117
C02980=1081.308,236.338,-79.661,175.233,24.478,154.116
C02981=1081.300,235.944,-79.619,175.229,24.472,154.115
C02982=1081.291,235.550,-79.578,175.224,24.467,154.115
C02983=1081.282,235.156,-79.536,175.221,24.462,154.114
C02984=1081.276,234.907,-79.510,175.219,24.459,154.114
C02985=1081.271,234.659,-79.483,175.216,24.455,154.114
C02986=1081.265,234.410,-79.456,175.214,24.452,154.113
C02987=1081.259,234.161,-79.430,175.210,24.449,154.113
C02988=1081.254,233.913,-79.404,175.208,24.445,154.112
C02989=1081.247,233.664,-79.378,175.206,24.442,154.112
C02990=1081.242,233.416,-79.352,175.203,24.439,154.112
C02991=1081.236,233.167,-79.326,175.201,24.436,154.111
C02992=1081.231,232.918,-79.300,175.199,24.432,154.111
C02993=1081.225,232.670,-79.273,175.196,24.429,154.110
C02994=1081.219,232.421,-79.247,175.194,24.426,154.110
C02995=1081.214,232.173,-79.222,175.191,24.422,154.110
C02996=1081.208,231.924,-79.196,175.189,24.419,154.109
C02997=1081.202,231.676,-79.169,175.187,24.416,154.109
C02998=1081.197,231.427,-79.143,175.183,24.412,154.108
C02999=1081.191,231.178,-79.117,175.181,24.409,154.108
C03000=1081.185,230.930,-79.091,175.179,24.406,154.108
C03001=1081.179,230.681,-79.065,175.176,24.402,154.107
C03002=1081.174,230.432,-79.039,175.174,24.399,154.107
C03003=1081.169,230.184,-79.013,175.171,24.395,154.106
C03004=1081.163,229.936,-78.988,175.169,24.392,154.106
C03005=1081.157,229.687,-78.962,175.167,24.389,154.106
C03006=1081.151,229.438,-78.935,175.164,24.385,154.105
C03007=1081.145,229.190,-78.910,175.162,24.382,154.105
C03008=1081.140,228.941,-78.884,175.160,24.379,154.104
C03009=1081.133,228.692,-78.859,175.157,24.375,154.104
C03010=1081.128,228.444,-78.832,175.154,24.372,154.104
C03011=1081.123,228.195,-78.806,175.152,24.369,154.103
C03012=1081.117,227.947,-78.781,175.149,24.366,154.103
C03013=1081.111,227.698,-78.755,175.147,24.362,154.102
C03014=1081.106,227.449,-78.729,175.145,24.359,154.102
C03015=1081.099,227.201,-78.703,175.142,24.356,154.102
C03016=1081.094,226.952,-78.677,175.140,24.353,154.101
C03017=1081.088,226.704,-78.652,175.138,24.350,154.101
C03018=1081.083,226.455,-78.626,175.135,24.346,154.101
C03019=1081.076,226.206,-78.601,175.132,24.343,154.100
C03020=1081.071,225.957,-78.575,175.130,24.340,154.100
C03021=1081.065,225.708,-78.549,175.127,24.336,154.099
C03022=1081.060,225.460,-78.524,175.125,24.333,154.099
C03023=1081.054,225.211,-78.498,175.123,24.330,154.098
C03024=1081.048,224.963,-78.473,175.120,24.326,154.098
C03025=1081.043,224.714,-78.447,175.118,24.323,154.098
C03026=1081.037,224.466,-78.421,175.116,24.320,154.097
C03027=1081.031,224.217,-78.395,175.113,24.316,154.097
C03028=1081.025,223.969,-78.370,175.111,24.313,154.097
C03029=1081.020,223.720,-78.344,175.109,24.310,154.096
C03030=1081.014,223.472,-78.319,175.106,24.306,154.096
C03031=1081.009,223.222,-78.294,175.103,24.303,154.095
C03032=1081.000,222.820,-78.252,175.100,24.297,154.095
C03033=1080.991,222.417,-78.211,175.095,24.292,154.094
C03034=1080.981,222.015,-78.170,175.092,24.287,154.093
C03035=1080.972,221.613,-78.128,175.088,24.282,154.093
C03036=1080.966,221.365,-78.103,175.085,24.278,154.092
C03037=1080.961,221.115,-78.078,175.083,24.275,154.092
C03038=1080.955,220.867,-78.053,175.081,24.272,154.092
C03039=1080.949,220.618,-78.028,175.079,24.268,154.091
C03040=1080.944,220.370,-78.002,175.076,24.265,154.091
C03041=1080.938,220.121,-77.977,175.074,24.262,154.090
C03042=1080.931,219.873,-77.951,175.072,24.259,154.090
C03043=1080.927,219.624,-77.927,175.069,24.255,154.090
C03044=1080.921,219.375,-77.901,175.067,24.252,154.089
C03045=1080.914,219.126,-77.876,175.064,24.249,154.089
C03046=1080.910,218.878,-77.850,175.062,24.246,154.088
C03047=1080.904,218.629,-77.826,175.059,24.242,154.088
C03048=1080.897,218.380,-77.800,175.057,24.239,154.088
C03049=1080.892,218.132,-77.775,175.055,24.236,154.087
C03050=1080.886,217.883,-77.749,175.052,24.232,154.087
C03051=1080.881,217.634,-77.725,175.050,24.229,154.086
C03052=1080.875,217.386,-77.700,175.048,24.226,154.086
C03053=1080.869,217.137,-77.674,175.046,24.222,154.086
C03054=1080.864,216.888,-77.650,175.043,24.219,154.085
C03055=1080.858,216.640,-77.624,175.041,24.216,154.085
C03056=1080.852,216.390,-77.600,175.039,24.212,154.084
C03057=1080.846,216.142,-77.575,175.036,24.209,154.084
C03058=1080.841,215.893,-77.549,175.033,24.206,154.084
C03059=1080.836,215.645,-77.524,175.031,24.202,154.083
C03060=1080.829,215.396,-77.499,175.029,24.199,154.083
C03061=1080.824,215.148,-77.475,175.026,24.196,154.083
C03062=1080.819,214.899,-77.449,175.024,24.192,154.082
C03063=1080.813,214.650,-77.425,175.022,24.189,154.082
C03064=1080.807,214.401,-77.399,175.020,24.186,154.081
C03065=1080.801,214.153,-77.374,175.017,24.182,154.081
C03066=1080.796,213.904,-77.350,175.015,24.179,154.080
C03067=1080.790,213.655,-77.324,175.013,24.176,154.080
C03068=1080.785,213.406,-77.300,175.011,24.173,154.080
C03069=1080.779,213.157,-77.275,175.008,24.169,154.079
C03070=1080.773,212.909,-77.250,175.006,24.166,154.079
C03071=1080.768,212.660,-77.225,175.003,24.163,154.078
C03072=1080.762,212.412,-77.200,175.001,24.160,154.078
C03073=1080.756,212.163,-77.176,174.998,24.156,154.078
C03074=1080.750,211.915,-77.151,174.996,24.153,154.077
C03075=1080.745,211.665,-77.126,174.994,24.150,154.077
C03076=1080.739,211.417,-77.102,174.992,24.147,154.077
C03077=1080.733,211.168,-77.077,174.989,24.143,154.076
C03078=1080.728,210.920,-77.052,174.987,24.140,154.076
C03079=1080.722,210.670,-77.028,174.985,24.137,154.075
C03080=1080.716,210.422,-77.003,174.983,24.134,154.075
C03081=1080.710,210.173,-76.978,174.980,24.130,154.075
C03082=1080.705,209.924,-76.954,174.977,24.127,154.074
C03083=1080.699,209.676,-76.929,174.975,24.124,154.074
C03084=1080.690,209.278,-76.889,174.972,24.118,154.073
C03085=1080.681,208.880,-76.850,174.968,24.113,154.073
C03086=1080.672,208.481,-76.810,174.965,24.108,154.072
C03087=1080.663,208.083,-76.771,174.960,24.103,154.071
C03088=1080.639,207.049,-76.672,174.863,24.050,154.073
C03089=1080.634,206.801,-76.648,174.859,24.047,154.073
C03090=1080.629,206.552,-76.623,174.857,24.045,154.073
C03091=1080.622,206.303,-76.599,174.854,24.043,154.073
C03092=1080.617,206.054,-76.576,174.852,24.040,154.072
C03093=1080.612,205.806,-76.551,174.850,24.038,154.072
C03094=1080.606,205.557,-76.528,174.847,24.036,154.072
C03095=1080.600,205.307,-76.504,174.845,24.034,154.072
C03096=1080.595,205.059,-76.480,174.843,24.031,154.072
C03097=1080.589,204.810,-76.456,174.840,24.029,154.072
C03098=1080.584,204.562,-76.432,174.838,24.027,154.071
C03099=1080.579,204.313,-76.408,174.836,24.025,154.071
C03100=1080.573,204.064,-76.385,174.833,24.022,154.071
C03101=1080.567,203.815,-76.360,174.831,24.020,154.071
C03102=1080.562,203.566,-76.336,174.828,24.017,154.071
C03103=1080.556,203.318,-76.313,174.826,24.015,154.071
C03104=1080.550,203.069,-76.288,174.824,24.013,154.070
C03105=1080.545,202.820,-76.265,174.821,24.010,154.070
C03106=1080.539,202.572,-76.241,174.818,24.008,154.070
C03107=1080.534,202.322,-76.217,174.816,24.006,154.070
C03108=1080.528,202.073,-76.194,174.813,24.003,154.070
C03109=1080.522,201.825,-76.170,174.811,24.001,154.069
C03110=1080.517,201.576,-76.146,174.809,23.998,154.069
C03111=1080.511,201.328,-76.123,174.806,23.996,154.069
C03112=1080.506,201.078,-76.099,174.804,23.994,154.069
C03113=1080.499,200.829,-76.075,174.801,23.992,154.069
C03114=1080.493,200.581,-76.052,174.799,23.990,154.069
C03115=1080.488,200.332,-76.028,174.797,23.987,154.069
C03116=1080.482,200.083,-76.005,174.794,23.985,154.068
C03117=1080.477,199.834,-75.981,174.792,23.983,154.068
C03118=1080.471,199.586,-75.958,174.790,23.980,154.068
C03119=1080.465,199.337,-75.934,174.787,23.978,154.068
C03120=1080.460,199.087,-75.910,174.785,23.976,154.068
C03121=1080.454,198.838,-75.887,174.782,23.974,154.068
C03122=1080.448,198.590,-75.864,174.780,23.972,154.067
C03123=1080.443,198.341,-75.840,174.778,23.969,154.067
C03124=1080.437,198.093,-75.817,174.775,23.967,154.067
C03125=1080.431,197.844,-75.794,174.773,23.964,154.067
C03126=1080.426,197.595,-75.770,174.771,23.962,154.067
C03127=1080.420,197.346,-75.746,174.768,23.960,154.067
C03128=1080.414,197.097,-75.723,174.766,23.958,154.066
C03129=1080.408,196.848,-75.699,174.763,23.956,154.066
C03130=1080.403,196.599,-75.676,174.761,23.953,154.066
C03131=1080.397,196.350,-75.653,174.759,23.951,154.066
C03132=1080.392,196.101,-75.629,174.756,23.949,154.066
C03133=1080.386,195.853,-75.606,174.754,23.946,154.066
C03134=1080.380,195.604,-75.583,174.752,23.944,154.065
C03135=1080.375,195.355,-75.559,174.749,23.942,154.065
C03136=1080.369,195.107,-75.536,174.747,23.939,154.065
C03137=1080.363,194.858,-75.513,174.745,23.937,154.065
C03138=1080.358,194.608,-75.489,174.742,23.935,154.065
C03139=1080.353,194.359,-75.466,174.740,23.933,154.065
C03140=1080.347,194.111,-75.442,174.737,23.930,154.065
C03141=1080.341,193.862,-75.420,174.735,23.928,154.064
C03142=1080.336,193.613,-75.396,174.733,23.926,154.064
C03143=1080.330,193.364,-75.373,174.730,23.923,154.064
C03144=1080.324,193.115,-75.350,174.729,23.922,154.064
C03145=1080.318,192.867,-75.326,174.726,23.919,154.064
C03146=1080.313,192.618,-75.303,174.724,23.917,154.063
C03147=1080.308,192.369,-75.280,174.722,23.914,154.063
C03148=1080.302,192.120,-75.257,174.719,23.912,154.063
C03149=1080.296,191.841,-75.231,174.716,23.910,154.063
C03150=1080.290,191.561,-75.205,174.714,23.907,154.063
C03151=1080.284,191.281,-75.179,174.711,23.905,154.063
C03152=1080.277,191.001,-75.153,174.708,23.902,154.062
C03153=1080.272,190.752,-75.130,174.707,23.900,154.062
C03154=1080.266,190.504,-75.107,174.704,23.898,154.062
C03155=1080.261,190.254,-75.084,174.702,23.895,154.062
C03156=1080.255,190.005,-75.061,174.700,23.893,154.062
C03157=1080.250,189.757,-75.038,174.697,23.890,154.061
C03158=1080.244,189.508,-75.015,174.695,23.888,154.061
C03159=1080.239,189.260,-74.992,174.693,23.885,154.061
C03160=1080.234,189.010,-74.969,174.690,23.883,154.061
C03161=1080.228,188.761,-74.946,174.688,23.881,154.061
C03162=1080.222,188.513,-74.923,174.686,23.879,154.061
C03163=1080.217,188.264,-74.900,174.683,23.876,154.060
C03164=1080.211,188.015,-74.877,174.681,23.874,154.060
C03165=1080.206,187.765,-74.853,174.679,23.872,154.060
C03166=1080.201,187.517,-74.831,174.677,23.870,154.060
C03167=1080.195,187.268,-74.808,174.675,23.867,154.060
C03168=1080.189,187.020,-74.785,174.673,23.865,154.059
C03169=1080.183,186.771,-74.762,174.670,23.863,154.059
C03170=1080.178,186.521,-74.738,174.668,23.860,154.059
C03171=1080.173,186.273,-74.715,174.665,23.858,154.059
C03172=1080.168,186.024,-74.693,174.663,23.856,154.059
C03173=1080.162,185.775,-74.670,174.661,23.853,154.059
C03174=1080.156,185.526,-74.648,174.658,23.851,154.058
C03175=1080.151,185.277,-74.625,174.656,23.849,154.058
C03176=1080.145,185.028,-74.602,174.654,23.846,154.058
C03177=1080.140,184.780,-74.579,174.652,23.844,154.058
C03178=1080.134,184.531,-74.556,174.650,23.842,154.058
C03179=1080.129,184.282,-74.534,174.647,23.840,154.058
C03180=1080.123,184.033,-74.511,174.645,23.838,154.057
C03181=1080.116,183.784,-74.489,174.643,23.835,154.057
C03182=1080.111,183.535,-74.466,174.640,23.833,154.057
C03183=1080.105,183.286,-74.443,174.638,23.831,154.057
C03184=1080.100,183.037,-74.421,174.636,23.829,154.057
C03185=1080.094,182.788,-74.398,174.634,23.827,154.057
C03186=1080.087,182.539,-74.375,174.632,23.824,154.056
C03187=1080.083,182.290,-74.353,174.629,23.822,154.056
C03188=1080.077,182.042,-74.330,174.627,23.820,154.056
C03189=1080.071,181.793,-74.307,174.625,23.818,154.056
C03190=1080.065,181.543,-74.286,174.622,23.816,154.056
C03191=1080.059,181.295,-74.263,174.620,23.813,154.056
C03192=1080.054,181.046,-74.240,174.617,23.811,154.056
C03193=1080.048,180.796,-74.218,174.616,23.809,154.055
C03194=1080.042,180.548,-74.196,174.614,23.807,154.055
C03195=1080.036,180.299,-74.173,174.611,23.804,154.055
C03196=1080.031,180.050,-74.151,174.609,23.802,154.055
C03197=1080.025,179.801,-74.128,174.607,23.800,154.055
C03198=1080.019,179.552,-74.106,174.604,23.798,154.055
C03199=1080.014,179.304,-74.083,174.602,23.796,154.054
C03200=1080.008,179.055,-74.060,174.600,23.794,154.054
C03201=1080.002,178.805,-74.039,174.598,23.792,154.054
C03202=1079.996,178.557,-74.016,174.596,23.789,154.054
C03203=1079.991,178.307,-73.994,174.593,23.787,154.054
C03204=1079.985,178.059,-73.972,174.591,23.784,154.054
C03205=1079.980,177.810,-73.949,174.589,23.782,154.053
C03206=1079.974,177.561,-73.926,174.587,23.780,154.053
C03207=1079.968,177.311,-73.905,174.585,23.778,154.053
C03208=1079.963,177.063,-73.882,174.582,23.776,154.053
C03209=1079.957,176.814,-73.860,174.580,23.774,154.053
C03210=1079.951,176.565,-73.838,174.577,23.772,154.053
C03211=1079.945,176.316,-73.815,174.575,23.769,154.052
C03212=1079.940,176.067,-73.793,174.574,23.767,154.052
C03213=1079.933,175.787,-73.768,174.570,23.764,154.052
C03214=1079.927,175.507,-73.743,174.568,23.762,154.052
C03215=1079.921,175.227,-73.718,174.566,23.759,154.052
C03216=1079.915,174.947,-73.694,174.564,23.757,154.052
C03217=1079.909,174.698,-73.671,174.561,23.754,154.051
C03218=1079.903,174.449,-73.649,174.559,23.752,154.051
C03219=1079.898,174.200,-73.627,174.557,23.750,154.051
C03220=1079.892,173.951,-73.604,174.555,23.748,154.051
C03221=1079.886,173.702,-73.582,174.553,23.746,154.051
C03222=1079.881,173.453,-73.561,174.550,23.743,154.051
C03223=1079.876,173.205,-73.538,174.548,23.741,154.050
C03224=1079.869,172.955,-73.516,174.546,23.739,154.050
C03225=1079.865,172.707,-73.494,174.544,23.737,154.050
C03226=1079.858,172.458,-73.472,174.542,23.734,154.050
C03227=1079.853,172.208,-73.450,174.540,23.732,154.050
C03228=1079.848,171.960,-73.428,174.537,23.730,154.050
C03229=1079.842,171.710,-73.406,174.535,23.728,154.049
C03230=1079.836,171.461,-73.383,174.533,23.726,154.049
C03231=1079.830,171.213,-73.362,174.531,23.723,154.049
C03232=1079.825,170.963,-73.340,174.529,23.721,154.049
C03233=1079.820,170.715,-73.318,174.526,23.719,154.049
C03234=1079.814,170.466,-73.295,174.525,23.717,154.048
C03235=1079.808,170.217,-73.273,174.523,23.714,154.048
C03236=1079.803,169.968,-73.252,174.520,23.712,154.048
C03237=1079.797,169.719,-73.230,174.518,23.710,154.048
C03238=1079.792,169.470,-73.208,174.515,23.707,154.048
C03239=1079.786,169.221,-73.186,174.514,23.705,154.047
C03240=1079.781,168.972,-73.164,174.512,23.703,154.047
C03241=1079.775,168.723,-73.142,174.509,23.701,154.047
C03242=1079.770,168.474,-73.120,174.507,23.698,154.047
C03243=1079.764,168.225,-73.098,174.506,23.696,154.047
C03244=1079.759,167.976,-73.076,174.503,23.694,154.047
C03245=1079.753,167.727,-73.055,174.501,23.692,154.046
C03246=1079.748,167.478,-73.033,174.499,23.689,154.046
C03247=1079.742,167.229,-73.011,174.496,23.687,154.046
C03248=1079.737,166.980,-72.989,174.495,23.685,154.046
C03249=1079.731,166.731,-72.968,174.493,23.682,154.046
C03250=1079.725,166.482,-72.945,174.490,23.680,154.046
C03251=1079.720,166.234,-72.924,174.488,23.678,154.045
C03252=1079.714,165.984,-72.902,174.486,23.676,154.045
C03253=1079.709,165.736,-72.880,174.484,23.673,154.045
C03254=1079.703,165.486,-72.858,174.482,23.671,154.045
C03255=1079.698,165.238,-72.837,174.479,23.669,154.045
C03256=1079.693,164.989,-72.815,174.478,23.666,154.044
C03257=1079.687,164.740,-72.793,174.476,23.664,154.044
C03258=1079.682,164.491,-72.771,174.473,23.662,154.044
C03259=1079.676,164.242,-72.750,174.472,23.659,154.044
C03260=1079.671,163.992,-72.729,174.470,23.657,154.044
C03261=1079.665,163.743,-72.707,174.467,23.655,154.043
C03262=1079.660,163.494,-72.685,174.465,23.652,154.043
C03263=1079.654,163.245,-72.663,174.464,23.650,154.043
C03264=1079.649,162.996,-72.642,174.461,23.648,154.043
C03265=1079.644,162.748,-72.620,174.459,23.645,154.043
C03266=1079.638,162.498,-72.598,174.457,23.643,154.043
C03267=1079.633,162.250,-72.577,174.455,23.641,154.042
C03268=1079.627,162.000,-72.555,174.453,23.639,154.042
C03269=1079.622,161.752,-72.533,174.451,23.636,154.042
C03270=1079.617,161.502,-72.512,174.448,23.634,154.042
C03271=1079.611,161.253,-72.491,174.447,23.632,154.041
C03272=1079.606,161.004,-72.469,174.445,23.630,154.041
C03273=1079.599,160.755,-72.448,174.442,23.627,154.041
C03274=1079.594,160.507,-72.426,174.441,23.625,154.041
C03275=1079.589,160.257,-72.405,174.438,23.623,154.041
C03276=1079.583,160.008,-72.384,174.436,23.621,154.041
C03277=1079.577,159.728,-72.360,174.434,23.618,154.040
C03278=1079.570,159.447,-72.335,174.431,23.616,154.040
C03279=1079.563,159.167,-72.311,174.429,23.613,154.040
C03280=1079.557,158.887,-72.288,174.427,23.611,154.040
C03281=1079.552,158.638,-72.266,174.425,23.608,154.040
C03282=1079.546,158.389,-72.244,174.423,23.606,154.039
C03283=1079.541,158.139,-72.224,174.421,23.604,154.039
C03284=1079.535,157.890,-72.202,174.418,23.602,154.039
C03285=1079.529,157.642,-72.181,174.417,23.599,154.039
C03286=1079.524,157.393,-72.160,174.415,23.597,154.039
C03287=1079.518,157.143,-72.138,174.412,23.595,154.039
C03288=1079.512,156.895,-72.117,174.410,23.593,154.038
C03289=1079.507,156.645,-72.096,174.409,23.590,154.038
C03290=1079.502,156.396,-72.074,174.406,23.588,154.038
C03291=1079.496,156.148,-72.053,174.404,23.586,154.038
C03292=1079.490,155.898,-72.032,174.403,23.583,154.038
C03293=1079.485,155.649,-72.011,174.400,23.581,154.037
C03294=1079.479,155.400,-71.990,174.398,23.579,154.037
C03295=1079.473,155.151,-71.969,174.396,23.577,154.037
C03296=1079.468,154.903,-71.947,174.394,23.574,154.037
C03297=1079.462,154.653,-71.927,174.392,23.572,154.037
C03298=1079.456,154.404,-71.905,174.390,23.570,154.037
C03299=1079.451,154.155,-71.885,174.388,23.568,154.036
C03300=1079.445,153.906,-71.863,174.386,23.565,154.036
C03301=1079.440,153.657,-71.843,174.384,23.563,154.036
C03302=1079.434,153.408,-71.821,174.382,23.561,154.036
C03303=1079.428,153.158,-71.800,174.380,23.559,154.036
C03304=1079.423,152.910,-71.779,174.378,23.557,154.035
C03305=1079.417,152.661,-71.759,174.376,23.554,154.035
C03306=1079.411,152.412,-71.737,174.374,23.552,154.035
C03307=1079.406,152.163,-71.716,174.372,23.550,154.035
C03308=1079.400,151.914,-71.695,174.370,23.548,154.035
C03309=1079.394,151.664,-71.674,174.368,23.545,154.035
C03310=1079.389,151.416,-71.653,174.366,23.543,154.034
C03311=1079.384,151.167,-71.632,174.364,23.541,154.034
C03312=1079.377,150.917,-71.611,174.361,23.539,154.034
C03313=1079.372,150.668,-71.590,174.360,23.536,154.034
C03314=1079.367,150.419,-71.570,174.358,23.534,154.034
C03315=1079.361,150.170,-71.548,174.355,23.532,154.033
C03316=1079.356,149.921,-71.527,174.354,23.529,154.033
C03317=1079.350,149.672,-71.506,174.352,23.527,154.033
C03318=1079.345,149.423,-71.486,174.349,23.525,154.033
C03319=1079.339,149.173,-71.465,174.348,23.523,154.033
C03320=1079.333,148.925,-71.444,174.346,23.520,154.032
C03321=1079.327,148.676,-71.423,174.344,23.518,154.032
C03322=1079.321,148.426,-71.403,174.342,23.516,154.032
C03323=1079.316,148.178,-71.381,174.340,23.513,154.032
C03324=1079.311,147.929,-71.361,174.338,23.512,154.032
C03325=1079.305,147.679,-71.340,174.336,23.509,154.031
C03326=1079.299,147.430,-71.320,174.334,23.507,154.031
C03327=1079.293,147.181,-71.299,174.332,23.505,154.031
C03328=1079.288,146.932,-71.278,174.330,23.503,154.031
C03329=1079.283,146.683,-71.257,174.328,23.500,154.031
C03330=1079.276,146.434,-71.236,174.326,23.498,154.030
C03331=1079.271,146.185,-71.216,174.324,23.496,154.030
C03332=1079.265,145.936,-71.195,174.322,23.493,154.030
C03333=1079.260,145.687,-71.175,174.320,23.491,154.030
C03334=1079.253,145.437,-71.154,174.318,23.489,154.030
C03335=1079.248,145.189,-71.133,174.316,23.487,154.029
C03336=1079.243,144.940,-71.113,174.314,23.484,154.029
C03337=1079.237,144.691,-71.092,174.313,23.482,154.029
C03338=1079.231,144.441,-71.072,174.310,23.480,154.029
C03339=1079.226,144.192,-71.051,174.308,23.477,154.029
C03340=1079.220,143.943,-71.031,174.307,23.476,154.029
C03341=1079.214,143.663,-71.007,174.304,23.473,154.028
C03342=1079.207,143.382,-70.984,174.302,23.470,154.028
C03343=1079.201,143.101,-70.961,174.300,23.468,154.028
C03344=1079.195,142.821,-70.938,174.298,23.465,154.028
C03345=1079.189,142.572,-70.918,174.295,23.463,154.028
C03346=1079.184,142.323,-70.897,174.294,23.460,154.027
C03347=1079.178,142.073,-70.876,174.292,23.458,154.027
C03348=1079.172,141.825,-70.856,174.290,23.456,154.027
C03349=1079.166,141.575,-70.835,174.288,23.454,154.027
C03350=1079.161,141.326,-70.814,174.286,23.451,154.027
C03351=1079.155,141.078,-70.794,174.284,23.449,154.026
C03352=1079.150,140.828,-70.774,174.282,23.447,154.026
C03353=1079.145,140.579,-70.753,174.281,23.444,154.026
C03354=1079.138,140.330,-70.733,174.278,23.442,154.026
C03355=1079.133,140.081,-70.713,174.276,23.440,154.026
C03356=1079.127,139.831,-70.692,174.275,23.438,154.025
C03357=1079.122,139.583,-70.672,174.272,23.435,154.025
C03358=1079.116,139.334,-70.651,174.271,23.433,154.025
C03359=1079.110,139.085,-70.631,174.269,23.431,154.025
C03360=1079.105,138.836,-70.611,174.266,23.428,154.025
C03361=1079.098,138.586,-70.591,174.265,23.426,154.024
C03362=1079.093,138.337,-70.570,174.263,23.424,154.024
C03363=1079.087,138.088,-70.551,174.261,23.422,154.024
C03364=1079.082,137.838,-70.530,174.259,23.419,154.024
C03365=1079.076,137.590,-70.510,174.257,23.417,154.023
C03366=1079.071,137.340,-70.490,174.255,23.415,154.023
C03367=1079.065,137.092,-70.470,174.253,23.412,154.023
C03368=1079.060,136.843,-70.449,174.251,23.411,154.023
C03369=1079.053,136.593,-70.429,174.249,23.408,154.023
C03370=1079.048,136.344,-70.408,174.248,23.406,154.022
C03371=1079.042,136.095,-70.388,174.245,23.404,154.022
C03372=1079.037,135.845,-70.369,174.244,23.401,154.022
C03373=1079.031,135.597,-70.349,174.242,23.399,154.022
C03374=1079.026,135.347,-70.328,174.240,23.397,154.022
C03375=1079.020,135.099,-70.308,174.238,23.394,154.021
C03376=1079.014,134.849,-70.288,174.236,23.392,154.021
C03377=1079.009,134.600,-70.268,174.234,23.390,154.021
C03378=1079.003,134.351,-70.248,174.232,23.388,154.021
C03379=1078.997,134.102,-70.228,174.231,23.385,154.021
C03380=1078.992,133.853,-70.207,174.228,23.383,154.020
C03381=1078.986,133.604,-70.187,174.227,23.381,154.020
C03382=1078.981,133.355,-70.168,174.225,23.378,154.020
C03383=1078.975,133.106,-70.147,174.223,23.376,154.020
C03384=1078.969,132.857,-70.127,174.221,23.374,154.020
C03385=1078.964,132.606,-70.107,174.219,23.371,154.019
C03386=1078.958,132.358,-70.087,174.217,23.369,154.019
C03387=1078.952,132.108,-70.067,174.215,23.367,154.019
C03388=1078.946,131.860,-70.047,174.214,23.364,154.019
C03389=1078.941,131.610,-70.028,174.211,23.362,154.019
C03390=1078.935,131.361,-70.008,174.210,23.360,154.018
C03391=1078.929,131.113,-69.988,174.208,23.358,154.018
C03392=1078.924,130.863,-69.968,174.206,23.356,154.018
C03393=1078.918,130.614,-69.948,174.204,23.353,154.018
C03394=1078.912,130.365,-69.928,174.203,23.351,154.018
C03395=1078.906,130.116,-69.909,174.200,23.349,154.017
C03396=1078.901,129.867,-69.888,174.198,23.346,154.017
C03397=1078.895,129.617,-69.869,174.197,23.344,154.017
C03398=1078.889,129.368,-69.849,174.194,23.342,154.017
C03399=1078.883,129.120,-69.829,174.193,23.340,154.017
C03400=1078.878,128.870,-69.810,174.191,23.337,154.016
C03401=1078.872,128.621,-69.790,174.189,23.335,154.016
C03402=1078.867,128.372,-69.770,174.187,23.333,154.016
C03403=1078.861,128.123,-69.750,174.186,23.331,154.016
C03404=1078.855,127.873,-69.731,174.183,23.328,154.016
C03405=1078.848,127.593,-69.708,174.181,23.325,154.015
C03406=1078.842,127.312,-69.686,174.180,23.324,154.015
C03407=1078.835,127.031,-69.663,174.178,23.321,154.015
C03408=1078.828,126.750,-69.642,174.175,23.318,154.015
C03409=1078.822,126.501,-69.622,174.173,23.316,154.015
C03410=1078.817,126.252,-69.602,174.172,23.313,154.014
C03411=1078.812,126.003,-69.582,174.169,23.311,154.014
C03412=1078.806,125.754,-69.563,174.168,23.309,154.014
C03413=1078.800,125.505,-69.543,174.166,23.306,154.014
C03414=1078.795,125.256,-69.524,174.164,23.304,154.013
C03415=1078.789,125.007,-69.504,174.162,23.302,154.013
C03416=1078.783,124.757,-69.485,174.161,23.299,154.013
C03417=1078.778,124.508,-69.465,174.158,23.297,154.013
C03418=1078.772,124.259,-69.445,174.157,23.295,154.013
C03419=1078.766,124.009,-69.426,174.155,23.293,154.012
C03420=1078.760,123.761,-69.406,174.153,23.291,154.012
C03421=1078.755,123.511,-69.386,174.151,23.288,154.012
C03422=1078.749,123.262,-69.367,174.150,23.286,154.012
C03423=1078.743,123.013,-69.347,174.147,23.283,154.011
C03424=1078.737,122.764,-69.328,174.146,23.281,154.011
C03425=1078.733,122.515,-69.309,174.144,23.279,154.011
C03426=1078.727,122.266,-69.289,174.143,23.276,154.011
C03427=1078.721,122.016,-69.269,174.140,23.274,154.011
C03428=1078.716,121.767,-69.250,174.139,23.272,154.010
C03429=1078.710,121.518,-69.230,174.137,23.269,154.010
C03430=1078.704,121.269,-69.211,174.135,23.267,154.010
C03431=1078.698,121.019,-69.192,174.133,23.265,154.010
C03432=1078.692,120.770,-69.172,174.132,23.262,154.009
C03433=1078.687,120.522,-69.153,174.129,23.260,154.009
C03434=1078.682,120.272,-69.134,174.128,23.258,154.009
C03435=1078.676,120.023,-69.114,174.126,23.255,154.009
C03436=1078.670,119.774,-69.094,174.124,23.253,154.009
C03437=1078.665,119.524,-69.074,174.123,23.251,154.008
C03438=1078.659,119.275,-69.055,174.121,23.248,154.008
C03439=1078.654,119.026,-69.036,174.119,23.246,154.008
C03440=1078.648,118.777,-69.017,174.117,23.244,154.008
C03441=1078.642,118.528,-68.997,174.116,23.241,154.007
C03442=1078.637,118.278,-68.978,174.114,23.239,154.007
C03443=1078.631,118.029,-68.959,174.112,23.237,154.007
C03444=1078.626,117.780,-68.940,174.110,23.234,154.007
C03445=1078.620,117.531,-68.921,174.109,23.232,154.007
C03446=1078.614,117.282,-68.901,174.106,23.229,154.006
C03447=1078.609,117.033,-68.881,174.105,23.227,154.006
C03448=1078.604,116.784,-68.862,174.103,23.225,154.006
C03449=1078.598,116.534,-68.843,174.101,23.222,154.006
C03450=1078.592,116.285,-68.824,174.099,23.220,154.005
C03451=1078.586,116.035,-68.805,174.098,23.218,154.005
C03452=1078.581,115.787,-68.786,174.096,23.215,154.005
C03453=1078.576,115.537,-68.767,174.094,23.212,154.005
C03454=1078.570,115.288,-68.747,174.093,23.211,154.004
C03455=1078.564,115.039,-68.727,174.091,23.208,154.004
C03456=1078.559,114.790,-68.709,174.089,23.206,154.004
C03457=1078.553,114.541,-68.689,174.087,23.203,154.004
C03458=1078.548,114.291,-68.670,174.086,23.201,154.003
C03459=1078.542,114.042,-68.651,174.084,23.199,154.003
C03460=1078.537,113.793,-68.632,174.082,23.196,154.003
C03461=1078.530,113.544,-68.613,174.080,23.194,154.003
C03462=1078.525,113.295,-68.594,174.079,23.192,154.003
C03463=1078.519,113.045,-68.575,174.076,23.189,154.002
C03464=1078.513,112.796,-68.556,174.075,23.187,154.002
C03465=1078.508,112.547,-68.537,174.074,23.184,154.002
C03466=1078.502,112.298,-68.517,174.071,23.182,154.002
C03467=1078.496,112.049,-68.499,174.070,23.180,154.001
C03468=1078.490,111.799,-68.480,174.068,23.177,154.001
C03469=1078.485,111.519,-68.458,174.066,23.174,154.001
C03470=1078.477,111.238,-68.437,174.064,23.172,154.001
C03471=1078.472,110.957,-68.416,174.062,23.170,154.000
C03472=1078.465,110.676,-68.395,174.060,23.167,154.000
C03473=1078.459,110.427,-68.376,174.059,23.164,154.000
C03474=1078.454,110.178,-68.357,174.056,23.162,154.000
C03475=1078.447,109.929,-68.338,174.055,23.160,154.000
C03476=1078.442,109.679,-68.319,174.053,23.158,153.999
C03477=1078.437,109.430,-68.300,174.051,23.155,153.999
C03478=1078.430,109.181,-68.282,174.050,23.153,153.999
C03479=1078.425,108.931,-68.263,174.048,23.150,153.999
C03480=1078.420,108.683,-68.244,174.047,23.148,153.998
C03481=1078.413,108.434,-68.225,174.044,23.146,153.998
C03482=1078.408,108.184,-68.206,174.043,23.143,153.998
C03483=1078.402,107.935,-68.187,174.041,23.141,153.998
C03484=1078.396,107.686,-68.169,174.039,23.139,153.997
C03485=1078.391,107.436,-68.150,174.038,23.136,153.997
C03486=1078.385,107.187,-68.131,174.036,23.134,153.997
C03487=1078.379,106.938,-68.112,174.034,23.132,153.997
C03488=1078.373,106.689,-68.093,174.032,23.129,153.997
C03489=1078.368,106.439,-68.074,174.031,23.127,153.996
C03490=1078.362,106.191,-68.056,174.029,23.124,153.996
C03491=1078.357,105.941,-68.037,174.027,23.122,153.996
C03492=1078.350,105.692,-68.018,174.026,23.120,153.996
C03493=1078.345,105.443,-68.000,174.024,23.117,153.995
C03494=1078.340,105.193,-67.981,174.022,23.115,153.995
C03495=1078.333,104.944,-67.962,174.020,23.113,153.995
C03496=1078.328,104.695,-67.944,174.019,23.110,153.995
C03497=1078.323,104.445,-67.925,174.017,23.107,153.994
C03498=1078.317,104.197,-67.907,174.015,23.105,153.994
C03499=1078.312,103.947,-67.888,174.014,23.103,153.994
C03500=1078.305,103.698,-67.869,174.012,23.100,153.994
C03501=1078.300,103.449,-67.850,174.010,23.098,153.993
C03502=1078.295,103.199,-67.832,174.008,23.096,153.993
C03503=1078.288,102.950,-67.813,174.007,23.093,153.993
C03504=1078.283,102.701,-67.794,174.006,23.091,153.993
C03505=1078.277,102.451,-67.776,174.003,23.089,153.992
C03506=1078.272,102.203,-67.758,174.002,23.086,153.992
C03507=1078.265,101.953,-67.739,174.000,23.083,153.992
C03508=1078.261,101.704,-67.721,173.998,23.082,153.992
C03509=1078.255,101.455,-67.702,173.997,23.079,153.991
C03510=1078.249,101.205,-67.684,173.995,23.076,153.991
C03511=1078.244,100.956,-67.665,173.994,23.074,153.991
C03512=1078.238,100.706,-67.647,173.991,23.072,153.991
C03513=1078.232,100.458,-67.629,173.990,23.069,153.990
C03514=1078.226,100.209,-67.609,173.989,23.067,153.990
C03515=1078.220,99.959,-67.591,173.986,23.065,153.990
C03516=1078.215,99.710,-67.572,173.985,23.062,153.990
C03517=1078.209,99.460,-67.555,173.983,23.060,153.990
C03518=1078.203,99.212,-67.536,173.982,23.058,153.989
C03519=1078.198,98.962,-67.518,173.980,23.055,153.989
C03520=1078.191,98.713,-67.499,173.978,23.053,153.989
C03521=1078.186,98.464,-67.482,173.977,23.050,153.989
C03522=1078.180,98.214,-67.462,173.975,23.048,153.988
C03523=1078.174,97.965,-67.445,173.973,23.046,153.988
C03524=1078.169,97.716,-67.425,173.972,23.043,153.988
C03525=1078.163,97.467,-67.408,173.970,23.041,153.988
C03526=1078.157,97.217,-67.390,173.968,23.039,153.987
C03527=1078.151,96.968,-67.371,173.967,23.036,153.987
C03528=1078.146,96.719,-67.353,173.965,23.033,153.987
C03529=1078.140,96.469,-67.335,173.963,23.032,153.987
C03530=1078.135,96.220,-67.316,173.961,23.029,153.986
C03531=1078.128,95.971,-67.298,173.960,23.026,153.986
C03532=1078.123,95.722,-67.280,173.959,23.024,153.986
C03533=1078.117,95.441,-67.260,173.957,23.021,153.986
C03534=1078.109,95.160,-67.239,173.954,23.018,153.985
C03535=1078.104,94.880,-67.218,173.953,23.016,153.985
C03536=1078.097,94.599,-67.198,173.951,23.013,153.985
C03537=1078.092,94.350,-67.180,173.950,23.011,153.985
C03538=1078.085,94.100,-67.161,173.947,23.009,153.984
C03539=1078.081,93.851,-67.143,173.946,23.006,153.984
C03540=1078.075,93.601,-67.125,173.944,23.003,153.984
C03541=1078.069,93.353,-67.107,173.943,23.001,153.984
C03542=1078.063,93.103,-67.089,173.941,22.999,153.983
C03543=1078.058,92.854,-67.071,173.939,22.996,153.983
C03544=1078.051,92.605,-67.052,173.938,22.994,153.983
C03545=1078.046,92.356,-67.035,173.937,22.991,153.983
C03546=1078.041,92.106,-67.016,173.934,22.989,153.982
C03547=1078.035,91.857,-66.999,173.933,22.987,153.982
C03548=1078.029,91.608,-66.980,173.931,22.984,153.982
C03549=1078.024,91.358,-66.962,173.930,22.982,153.982
C03550=1078.018,91.109,-66.944,173.928,22.979,153.981
C03551=1078.012,90.859,-66.926,173.926,22.977,153.981
C03552=1078.007,90.610,-66.909,173.925,22.974,153.981
C03553=1078.000,90.361,-66.890,173.923,22.972,153.981
C03554=1077.995,90.112,-66.873,173.921,22.969,153.980
C03555=1077.989,89.862,-66.855,173.920,22.967,153.980
C03556=1077.983,89.613,-66.837,173.919,22.965,153.980
C03557=1077.978,89.363,-66.818,173.916,22.962,153.980
C03558=1077.972,89.115,-66.800,173.915,22.960,153.979
C03559=1077.966,88.865,-66.782,173.913,22.957,153.979
C03560=1077.960,88.616,-66.765,173.912,22.955,153.979
C03561=1077.954,88.366,-66.747,173.910,22.953,153.979
C03562=1077.949,88.117,-66.729,173.908,22.950,153.978
C03563=1077.943,87.868,-66.712,173.907,22.948,153.978
C03564=1077.937,87.619,-66.694,173.905,22.946,153.978
C03565=1077.931,87.370,-66.676,173.903,22.943,153.978
C03566=1077.925,87.120,-66.657,173.902,22.941,153.977
C03567=1077.919,86.871,-66.640,173.901,22.938,153.977
C03568=1077.913,86.622,-66.622,173.898,22.936,153.977
C03569=1077.908,86.373,-66.604,173.897,22.933,153.977
C03570=1077.902,86.124,-66.587,173.896,22.931,153.976
C03571=1077.896,85.874,-66.569,173.894,22.929,153.976
C03572=1077.891,85.625,-66.551,173.892,22.926,153.976
C03573=1077.885,85.375,-66.533,173.891,22.924,153.976
C03574=1077.880,85.126,-66.515,173.889,22.921,153.975
C03575=1077.874,84.877,-66.498,173.887,22.919,153.975
C03576=1077.868,84.627,-66.480,173.886,22.917,153.975
C03577=1077.863,84.378,-66.462,173.884,22.914,153.975
C03578=1077.857,84.129,-66.445,173.883,22.911,153.974
C03579=1077.851,83.879,-66.427,173.881,22.910,153.974
C03580=1077.845,83.630,-66.409,173.879,22.907,153.974
C03581=1077.839,83.380,-66.391,173.878,22.904,153.974
C03582=1077.834,83.131,-66.374,173.877,22.902,153.973
C03583=1077.828,82.882,-66.356,173.875,22.899,153.973
C03584=1077.822,82.632,-66.338,173.873,22.897,153.973
C03585=1077.817,82.383,-66.321,173.872,22.895,153.972
C03586=1077.811,82.134,-66.303,173.870,22.892,153.972
C03587=1077.805,81.885,-66.285,173.868,22.890,153.972
C03588=1077.800,81.636,-66.267,173.867,22.887,153.972
C03589=1077.794,81.386,-66.251,173.865,22.884,153.971
C03590=1077.789,81.137,-66.233,173.864,22.882,153.971
C03591=1077.783,80.887,-66.215,173.862,22.880,153.971
C03592=1077.777,80.638,-66.198,173.860,22.877,153.971
C03593=1077.771,80.389,-66.181,173.859,22.875,153.970
C03594=1077.765,80.140,-66.163,173.858,22.872,153.970
C03595=1077.759,79.891,-66.145,173.856,22.870,153.970
C03596=1077.754,79.641,-66.128,173.854,22.867,153.970
C03597=1077.749,79.417,-66.111,173.853,22.865,153.969
C03598=1077.744,79.193,-66.096,173.852,22.863,153.969
C03599=1077.739,78.968,-66.080,173.850,22.861,153.969
C03600=1077.733,78.743,-66.064,173.848,22.858,153.969
C03601=1077.729,78.519,-66.048,173.847,22.856,153.968
C03602=1077.723,78.294,-66.033,173.845,22.854,153.968
C03603=1077.718,78.071,-66.017,173.844,22.852,153.968
C03604=1077.713,77.846,-66.001,173.843,22.850,153.968
C03605=1077.707,77.596,-65.985,173.841,22.847,153.967
C03606=1077.701,77.347,-65.967,173.840,22.845,153.967
C03607=1077.695,77.098,-65.949,173.838,22.843,153.967
C03608=1077.690,76.849,-65.932,173.837,22.840,153.967
C03609=1077.685,76.599,-65.915,173.835,22.838,153.966
C03610=1077.678,76.349,-65.898,173.833,22.835,153.966
C03611=1077.672,76.100,-65.880,173.832,22.832,153.966
C03612=1077.667,75.851,-65.863,173.831,22.831,153.966
C03613=1077.661,75.602,-65.846,173.828,22.828,153.965
C03614=1077.655,75.352,-65.828,173.827,22.825,153.965
C03615=1077.649,75.103,-65.811,173.826,22.823,153.965
C03616=1077.644,74.854,-65.794,173.824,22.820,153.965
C03617=1077.636,74.524,-65.771,173.822,22.817,153.964
C03618=1077.628,74.193,-65.748,173.820,22.814,153.964
C03619=1077.621,73.862,-65.725,173.818,22.811,153.964
C03620=1077.613,73.532,-65.702,173.816,22.807,153.963
C03621=1077.608,73.282,-65.685,173.814,22.805,153.963
C03622=1077.602,73.033,-65.668,173.812,22.802,153.963
C03623=1077.596,72.783,-65.651,173.811,22.800,153.962
C03624=1077.590,72.534,-65.633,173.810,22.798,153.962
C03625=1077.584,72.285,-65.616,173.808,22.795,153.962
C03626=1077.579,72.036,-65.600,173.806,22.792,153.962
C03627=1077.573,71.787,-65.582,173.805,22.790,153.961
C03628=1077.567,71.536,-65.565,173.804,22.788,153.961
C03629=1077.561,71.288,-65.548,173.802,22.785,153.961
